   S706_TL_DC_3RD_CLAMP.Adv_End := TRUE;
   S706_TL_DC_3RD_CLAMP.Ret_End := FALSE;
   S706_TL_DC_U262_1_UP_DN.Enable_Aux := TRUE;
   S706_TL_DC_U262_1_UP_DN.Adv_Amount := 1;
   S706_TL_DC_U262_1_UP_DN.Ret_Amount := 1;
   S706_TL_DC_U262_1_UP_DN.LS_Adv1 := FALSE;
   S706_TL_DC_U262_1_UP_DN.LS_Ret1 := TRUE;
   S706_TL_DC_U262_1_UP_DN.LS_Adv2 := FALSE;
   S706_TL_DC_U262_1_UP_DN.LS_Ret2 := FALSE;
   S706_TL_DC_U262_1_UP_DN.LS_Adv3 := FALSE;
   S706_TL_DC_U262_1_UP_DN.LS_Ret3 := FALSE;
   S706_TL_DC_U262_1_UP_DN.LS_Adv4 := FALSE;
   S706_TL_DC_U262_1_UP_DN.LS_Ret4 := FALSE;
   S706_TL_DC_U262_1_UP_DN.LS_Adv5 := FALSE;
   S706_TL_DC_U262_1_UP_DN.LS_Ret5 := FALSE;
   S706_TL_DC_U262_1_UP_DN.LS_Adv6 := FALSE;
   S706_TL_DC_U262_1_UP_DN.LS_Ret6 := FALSE;
   S706_TL_DC_U262_1_UP_DN.LS_Adv7 := FALSE;
   S706_TL_DC_U262_1_UP_DN.LS_Ret7 := FALSE;
   S706_TL_DC_U262_1_UP_DN.LS_Adv8 := FALSE;
   S706_TL_DC_U262_1_UP_DN.LS_Ret8 := FALSE;
   S706_TL_DC_U262_1_UP_DN.SOL_Adv := FALSE;
   S706_TL_DC_U262_1_UP_DN.SOL_Ret := FALSE;
   S706_TL_DC_U262_1_UP_DN.M_Ready := TRUE;
   S706_TL_DC_U262_1_UP_DN.T_CHK1 := T#4S;
   S706_TL_DC_U262_1_UP_DN.T_CHK2 := T#4S;
   S706_TL_DC_U262_1_UP_DN.PB_Lamp_CHK := FALSE;
   S706_TL_DC_U262_1_UP_DN.PB_Error_Rst := FALSE;
   S706_TL_DC_U262_1_UP_DN.M_FLICK := FALSE;
   S706_TL_DC_U262_1_UP_DN.M_Adv_Err := FALSE;
   S706_TL_DC_U262_1_UP_DN.M_Ret_Err := FALSE;
   S706_TL_DC_U262_1_UP_DN.LP_Adv := FALSE;
   S706_TL_DC_U262_1_UP_DN.LP_Ret := TRUE;
   S706_TL_DC_U262_1_UP_DN.Visu_Adv := W#16#0;
   S706_TL_DC_U262_1_UP_DN.Visu_Ret := W#16#300;
   S706_TL_DC_U262_1_UP_DN.Error_T1.IN := FALSE;
   S706_TL_DC_U262_1_UP_DN.Error_T1.PT := T#4S;
   S706_TL_DC_U262_1_UP_DN.Error_T1.Q := FALSE;
   S706_TL_DC_U262_1_UP_DN.Error_T1.ET := T#0MS;
   S706_TL_DC_U262_1_UP_DN.Error_T1.STATE := B#16#0;
   S706_TL_DC_U262_1_UP_DN.Error_T1.STIME := T#23D5H8M21S546MS;
   S706_TL_DC_U262_1_UP_DN.Error_T1.ATIME := T#23D5H8M21S773MS;
   S706_TL_DC_U262_1_UP_DN.Error_T2.IN := FALSE;
   S706_TL_DC_U262_1_UP_DN.Error_T2.PT := T#4S;
   S706_TL_DC_U262_1_UP_DN.Error_T2.Q := FALSE;
   S706_TL_DC_U262_1_UP_DN.Error_T2.ET := T#0MS;
   S706_TL_DC_U262_1_UP_DN.Error_T2.STATE := B#16#0;
   S706_TL_DC_U262_1_UP_DN.Error_T2.STIME := T#0MS;
   S706_TL_DC_U262_1_UP_DN.Error_T2.ATIME := T#0MS;
   S706_TL_DC_U262_1_UP_DN.Adv_End_Aux := FALSE;
   S706_TL_DC_U262_1_UP_DN.Ret_End_Aux := TRUE;
   S706_TL_DC_U262_1_UP_DN.CHK_Aux1 := FALSE;
   S706_TL_DC_U262_1_UP_DN.CHK_Aux2 := FALSE;
   S706_TL_DC_U262_1_UP_DN.Error_T1_DN := FALSE;
   S706_TL_DC_U262_1_UP_DN.Error_T2_DN := FALSE;
   S706_TL_DC_U262_1_UP_DN.Adv_Memo := FALSE;
   S706_TL_DC_U262_1_UP_DN.Visu_Adv_Arr[0] := FALSE;
   S706_TL_DC_U262_1_UP_DN.Visu_Adv_Arr[1] := FALSE;
   S706_TL_DC_U262_1_UP_DN.Visu_Adv_Arr[2] := FALSE;
   S706_TL_DC_U262_1_UP_DN.Visu_Adv_Arr[3] := FALSE;
   S706_TL_DC_U262_1_UP_DN.Visu_Adv_Arr[4] := FALSE;
   S706_TL_DC_U262_1_UP_DN.Visu_Adv_Arr[5] := FALSE;
   S706_TL_DC_U262_1_UP_DN.Visu_Adv_Arr[6] := FALSE;
   S706_TL_DC_U262_1_UP_DN.Visu_Adv_Arr[7] := FALSE;
   S706_TL_DC_U262_1_UP_DN.Visu_Adv_Arr[8] := FALSE;
   S706_TL_DC_U262_1_UP_DN.Visu_Adv_Arr[9] := FALSE;
   S706_TL_DC_U262_1_UP_DN.Visu_Adv_Arr[10] := FALSE;
   S706_TL_DC_U262_1_UP_DN.Visu_Adv_Arr[11] := FALSE;
   S706_TL_DC_U262_1_UP_DN.Visu_Adv_Arr[12] := FALSE;
   S706_TL_DC_U262_1_UP_DN.Visu_Adv_Arr[13] := FALSE;
   S706_TL_DC_U262_1_UP_DN.Visu_Adv_Arr[14] := FALSE;
   S706_TL_DC_U262_1_UP_DN.Visu_Adv_Arr[15] := FALSE;
   S706_TL_DC_U262_1_UP_DN.Visu_Ret_Arr[0] := TRUE;
   S706_TL_DC_U262_1_UP_DN.Visu_Ret_Arr[1] := TRUE;
   S706_TL_DC_U262_1_UP_DN.Visu_Ret_Arr[2] := FALSE;
   S706_TL_DC_U262_1_UP_DN.Visu_Ret_Arr[3] := FALSE;
   S706_TL_DC_U262_1_UP_DN.Visu_Ret_Arr[4] := FALSE;
   S706_TL_DC_U262_1_UP_DN.Visu_Ret_Arr[5] := FALSE;
   S706_TL_DC_U262_1_UP_DN.Visu_Ret_Arr[6] := FALSE;
   S706_TL_DC_U262_1_UP_DN.Visu_Ret_Arr[7] := FALSE;
   S706_TL_DC_U262_1_UP_DN.Visu_Ret_Arr[8] := FALSE;
   S706_TL_DC_U262_1_UP_DN.Visu_Ret_Arr[9] := FALSE;
   S706_TL_DC_U262_1_UP_DN.Visu_Ret_Arr[10] := FALSE;
   S706_TL_DC_U262_1_UP_DN.Visu_Ret_Arr[11] := FALSE;
   S706_TL_DC_U262_1_UP_DN.Visu_Ret_Arr[12] := FALSE;
   S706_TL_DC_U262_1_UP_DN.Visu_Ret_Arr[13] := FALSE;
   S706_TL_DC_U262_1_UP_DN.Visu_Ret_Arr[14] := FALSE;
   S706_TL_DC_U262_1_UP_DN.Visu_Ret_Arr[15] := FALSE;
   S706_TL_DC_U262_1_UP_DN.BLK_Move_Ret := 0;
   S706_TL_DC_U262_1_UP_DN.Enable := TRUE;
   S706_TL_DC_U262_1_UP_DN.Adv_End := FALSE;
   S706_TL_DC_U262_1_UP_DN.Ret_End := TRUE;
   S706_TL_DC_U262_1.Enable_Aux := TRUE;
   S706_TL_DC_U262_1.Adv_Amount := 1;
   S706_TL_DC_U262_1.Ret_Amount := 1;
   S706_TL_DC_U262_1.LS_Adv1 := FALSE;
   S706_TL_DC_U262_1.LS_Ret1 := TRUE;
   S706_TL_DC_U262_1.LS_Adv2 := FALSE;
   S706_TL_DC_U262_1.LS_Ret2 := FALSE;
   S706_TL_DC_U262_1.LS_Adv3 := FALSE;
   S706_TL_DC_U262_1.LS_Ret3 := FALSE;
   S706_TL_DC_U262_1.LS_Adv4 := FALSE;
   S706_TL_DC_U262_1.LS_Ret4 := FALSE;
   S706_TL_DC_U262_1.LS_Adv5 := FALSE;
   S706_TL_DC_U262_1.LS_Ret5 := FALSE;
   S706_TL_DC_U262_1.LS_Adv6 := FALSE;
   S706_TL_DC_U262_1.LS_Ret6 := FALSE;
   S706_TL_DC_U262_1.LS_Adv7 := FALSE;
   S706_TL_DC_U262_1.LS_Ret7 := FALSE;
   S706_TL_DC_U262_1.LS_Adv8 := FALSE;
   S706_TL_DC_U262_1.LS_Ret8 := FALSE;
   S706_TL_DC_U262_1.SOL_Adv := FALSE;
   S706_TL_DC_U262_1.SOL_Ret := FALSE;
   S706_TL_DC_U262_1.M_Ready := TRUE;
   S706_TL_DC_U262_1.T_CHK1 := T#4S;
   S706_TL_DC_U262_1.T_CHK2 := T#4S;
   S706_TL_DC_U262_1.PB_Lamp_CHK := FALSE;
   S706_TL_DC_U262_1.PB_Error_Rst := FALSE;
   S706_TL_DC_U262_1.M_FLICK := FALSE;
   S706_TL_DC_U262_1.M_Adv_Err := FALSE;
   S706_TL_DC_U262_1.M_Ret_Err := FALSE;
   S706_TL_DC_U262_1.LP_Adv := FALSE;
   S706_TL_DC_U262_1.LP_Ret := TRUE;
   S706_TL_DC_U262_1.Visu_Adv := W#16#0;
   S706_TL_DC_U262_1.Visu_Ret := W#16#300;
   S706_TL_DC_U262_1.Error_T1.IN := FALSE;
   S706_TL_DC_U262_1.Error_T1.PT := T#4S;
   S706_TL_DC_U262_1.Error_T1.Q := FALSE;
   S706_TL_DC_U262_1.Error_T1.ET := T#0MS;
   S706_TL_DC_U262_1.Error_T1.STATE := B#16#0;
   S706_TL_DC_U262_1.Error_T1.STIME := T#23D2H56M52S237MS;
   S706_TL_DC_U262_1.Error_T1.ATIME := T#23D2H56M52S283MS;
   S706_TL_DC_U262_1.Error_T2.IN := FALSE;
   S706_TL_DC_U262_1.Error_T2.PT := T#4S;
   S706_TL_DC_U262_1.Error_T2.Q := FALSE;
   S706_TL_DC_U262_1.Error_T2.ET := T#0MS;
   S706_TL_DC_U262_1.Error_T2.STATE := B#16#0;
   S706_TL_DC_U262_1.Error_T2.STIME := T#0MS;
   S706_TL_DC_U262_1.Error_T2.ATIME := T#0MS;
   S706_TL_DC_U262_1.Adv_End_Aux := FALSE;
   S706_TL_DC_U262_1.Ret_End_Aux := TRUE;
   S706_TL_DC_U262_1.CHK_Aux1 := FALSE;
   S706_TL_DC_U262_1.CHK_Aux2 := FALSE;
   S706_TL_DC_U262_1.Error_T1_DN := FALSE;
   S706_TL_DC_U262_1.Error_T2_DN := FALSE;
   S706_TL_DC_U262_1.Adv_Memo := FALSE;
   S706_TL_DC_U262_1.Visu_Adv_Arr[0] := FALSE;
   S706_TL_DC_U262_1.Visu_Adv_Arr[1] := FALSE;
   S706_TL_DC_U262_1.Visu_Adv_Arr[2] := FALSE;
   S706_TL_DC_U262_1.Visu_Adv_Arr[3] := FALSE;
   S706_TL_DC_U262_1.Visu_Adv_Arr[4] := FALSE;
   S706_TL_DC_U262_1.Visu_Adv_Arr[5] := FALSE;
   S706_TL_DC_U262_1.Visu_Adv_Arr[6] := FALSE;
   S706_TL_DC_U262_1.Visu_Adv_Arr[7] := FALSE;
   S706_TL_DC_U262_1.Visu_Adv_Arr[8] := FALSE;
   S706_TL_DC_U262_1.Visu_Adv_Arr[9] := FALSE;
   S706_TL_DC_U262_1.Visu_Adv_Arr[10] := FALSE;
   S706_TL_DC_U262_1.Visu_Adv_Arr[11] := FALSE;
   S706_TL_DC_U262_1.Visu_Adv_Arr[12] := FALSE;
   S706_TL_DC_U262_1.Visu_Adv_Arr[13] := FALSE;
   S706_TL_DC_U262_1.Visu_Adv_Arr[14] := FALSE;
   S706_TL_DC_U262_1.Visu_Adv_Arr[15] := FALSE;
   S706_TL_DC_U262_1.Visu_Ret_Arr[0] := TRUE;
   S706_TL_DC_U262_1.Visu_Ret_Arr[1] := TRUE;
   S706_TL_DC_U262_1.Visu_Ret_Arr[2] := FALSE;
   S706_TL_DC_U262_1.Visu_Ret_Arr[3] := FALSE;
   S706_TL_DC_U262_1.Visu_Ret_Arr[4] := FALSE;
   S706_TL_DC_U262_1.Visu_Ret_Arr[5] := FALSE;
   S706_TL_DC_U262_1.Visu_Ret_Arr[6] := FALSE;
   S706_TL_DC_U262_1.Visu_Ret_Arr[7] := FALSE;
   S706_TL_DC_U262_1.Visu_Ret_Arr[8] := FALSE;
   S706_TL_DC_U262_1.Visu_Ret_Arr[9] := FALSE;
   S706_TL_DC_U262_1.Visu_Ret_Arr[10] := FALSE;
   S706_TL_DC_U262_1.Visu_Ret_Arr[11] := FALSE;
   S706_TL_DC_U262_1.Visu_Ret_Arr[12] := FALSE;
   S706_TL_DC_U262_1.Visu_Ret_Arr[13] := FALSE;
   S706_TL_DC_U262_1.Visu_Ret_Arr[14] := FALSE;
   S706_TL_DC_U262_1.Visu_Ret_Arr[15] := FALSE;
   S706_TL_DC_U262_1.BLK_Move_Ret := 0;
   S706_TL_DC_U262_1.Enable := TRUE;
   S706_TL_DC_U262_1.Adv_End := FALSE;
   S706_TL_DC_U262_1.Ret_End := TRUE;
   S706_TL_DC_U262_1_CLAMP.Enable_Aux := TRUE;
   S706_TL_DC_U262_1_CLAMP.Adv_Amount := 1;
   S706_TL_DC_U262_1_CLAMP.Ret_Amount := 1;
   S706_TL_DC_U262_1_CLAMP.LS_Adv1 := FALSE;
   S706_TL_DC_U262_1_CLAMP.LS_Ret1 := TRUE;
   S706_TL_DC_U262_1_CLAMP.LS_Adv2 := FALSE;
   S706_TL_DC_U262_1_CLAMP.LS_Ret2 := FALSE;
   S706_TL_DC_U262_1_CLAMP.LS_Adv3 := FALSE;
   S706_TL_DC_U262_1_CLAMP.LS_Ret3 := FALSE;
   S706_TL_DC_U262_1_CLAMP.LS_Adv4 := FALSE;
   S706_TL_DC_U262_1_CLAMP.LS_Ret4 := FALSE;
   S706_TL_DC_U262_1_CLAMP.LS_Adv5 := FALSE;
   S706_TL_DC_U262_1_CLAMP.LS_Ret5 := FALSE;
   S706_TL_DC_U262_1_CLAMP.LS_Adv6 := FALSE;
   S706_TL_DC_U262_1_CLAMP.LS_Ret6 := FALSE;
   S706_TL_DC_U262_1_CLAMP.LS_Adv7 := FALSE;
   S706_TL_DC_U262_1_CLAMP.LS_Ret7 := FALSE;
   S706_TL_DC_U262_1_CLAMP.LS_Adv8 := FALSE;
   S706_TL_DC_U262_1_CLAMP.LS_Ret8 := FALSE;
   S706_TL_DC_U262_1_CLAMP.SOL_Adv := FALSE;
   S706_TL_DC_U262_1_CLAMP.SOL_Ret := FALSE;
   S706_TL_DC_U262_1_CLAMP.M_Ready := TRUE;
   S706_TL_DC_U262_1_CLAMP.T_CHK1 := T#4S;
   S706_TL_DC_U262_1_CLAMP.T_CHK2 := T#4S;
   S706_TL_DC_U262_1_CLAMP.PB_Lamp_CHK := FALSE;
   S706_TL_DC_U262_1_CLAMP.PB_Error_Rst := FALSE;
   S706_TL_DC_U262_1_CLAMP.M_FLICK := FALSE;
   S706_TL_DC_U262_1_CLAMP.M_Adv_Err := FALSE;
   S706_TL_DC_U262_1_CLAMP.M_Ret_Err := FALSE;
   S706_TL_DC_U262_1_CLAMP.LP_Adv := FALSE;
   S706_TL_DC_U262_1_CLAMP.LP_Ret := TRUE;
   S706_TL_DC_U262_1_CLAMP.Visu_Adv := W#16#0;
   S706_TL_DC_U262_1_CLAMP.Visu_Ret := W#16#300;
   S706_TL_DC_U262_1_CLAMP.Error_T1.IN := FALSE;
   S706_TL_DC_U262_1_CLAMP.Error_T1.PT := T#4S;
   S706_TL_DC_U262_1_CLAMP.Error_T1.Q := FALSE;
   S706_TL_DC_U262_1_CLAMP.Error_T1.ET := T#0MS;
   S706_TL_DC_U262_1_CLAMP.Error_T1.STATE := B#16#0;
   S706_TL_DC_U262_1_CLAMP.Error_T1.STIME := T#23D2H56M52S237MS;
   S706_TL_DC_U262_1_CLAMP.Error_T1.ATIME := T#23D2H56M52S283MS;
   S706_TL_DC_U262_1_CLAMP.Error_T2.IN := FALSE;
   S706_TL_DC_U262_1_CLAMP.Error_T2.PT := T#4S;
   S706_TL_DC_U262_1_CLAMP.Error_T2.Q := FALSE;
   S706_TL_DC_U262_1_CLAMP.Error_T2.ET := T#0MS;
   S706_TL_DC_U262_1_CLAMP.Error_T2.STATE := B#16#0;
   S706_TL_DC_U262_1_CLAMP.Error_T2.STIME := T#0MS;
   S706_TL_DC_U262_1_CLAMP.Error_T2.ATIME := T#0MS;
   S706_TL_DC_U262_1_CLAMP.Adv_End_Aux := FALSE;
   S706_TL_DC_U262_1_CLAMP.Ret_End_Aux := TRUE;
   S706_TL_DC_U262_1_CLAMP.CHK_Aux1 := FALSE;
   S706_TL_DC_U262_1_CLAMP.CHK_Aux2 := FALSE;
   S706_TL_DC_U262_1_CLAMP.Error_T1_DN := FALSE;
   S706_TL_DC_U262_1_CLAMP.Error_T2_DN := FALSE;
   S706_TL_DC_U262_1_CLAMP.Adv_Memo := FALSE;
   S706_TL_DC_U262_1_CLAMP.Visu_Adv_Arr[0] := FALSE;
   S706_TL_DC_U262_1_CLAMP.Visu_Adv_Arr[1] := FALSE;
   S706_TL_DC_U262_1_CLAMP.Visu_Adv_Arr[2] := FALSE;
   S706_TL_DC_U262_1_CLAMP.Visu_Adv_Arr[3] := FALSE;
   S706_TL_DC_U262_1_CLAMP.Visu_Adv_Arr[4] := FALSE;
   S706_TL_DC_U262_1_CLAMP.Visu_Adv_Arr[5] := FALSE;
   S706_TL_DC_U262_1_CLAMP.Visu_Adv_Arr[6] := FALSE;
   S706_TL_DC_U262_1_CLAMP.Visu_Adv_Arr[7] := FALSE;
   S706_TL_DC_U262_1_CLAMP.Visu_Adv_Arr[8] := FALSE;
   S706_TL_DC_U262_1_CLAMP.Visu_Adv_Arr[9] := FALSE;
   S706_TL_DC_U262_1_CLAMP.Visu_Adv_Arr[10] := FALSE;
   S706_TL_DC_U262_1_CLAMP.Visu_Adv_Arr[11] := FALSE;
   S706_TL_DC_U262_1_CLAMP.Visu_Adv_Arr[12] := FALSE;
   S706_TL_DC_U262_1_CLAMP.Visu_Adv_Arr[13] := FALSE;
   S706_TL_DC_U262_1_CLAMP.Visu_Adv_Arr[14] := FALSE;
   S706_TL_DC_U262_1_CLAMP.Visu_Adv_Arr[15] := FALSE;
   S706_TL_DC_U262_1_CLAMP.Visu_Ret_Arr[0] := TRUE;
   S706_TL_DC_U262_1_CLAMP.Visu_Ret_Arr[1] := TRUE;
   S706_TL_DC_U262_1_CLAMP.Visu_Ret_Arr[2] := FALSE;
   S706_TL_DC_U262_1_CLAMP.Visu_Ret_Arr[3] := FALSE;
   S706_TL_DC_U262_1_CLAMP.Visu_Ret_Arr[4] := FALSE;
   S706_TL_DC_U262_1_CLAMP.Visu_Ret_Arr[5] := FALSE;
   S706_TL_DC_U262_1_CLAMP.Visu_Ret_Arr[6] := FALSE;
   S706_TL_DC_U262_1_CLAMP.Visu_Ret_Arr[7] := FALSE;
   S706_TL_DC_U262_1_CLAMP.Visu_Ret_Arr[8] := FALSE;
   S706_TL_DC_U262_1_CLAMP.Visu_Ret_Arr[9] := FALSE;
   S706_TL_DC_U262_1_CLAMP.Visu_Ret_Arr[10] := FALSE;
   S706_TL_DC_U262_1_CLAMP.Visu_Ret_Arr[11] := FALSE;
   S706_TL_DC_U262_1_CLAMP.Visu_Ret_Arr[12] := FALSE;
   S706_TL_DC_U262_1_CLAMP.Visu_Ret_Arr[13] := FALSE;
   S706_TL_DC_U262_1_CLAMP.Visu_Ret_Arr[14] := FALSE;
   S706_TL_DC_U262_1_CLAMP.Visu_Ret_Arr[15] := FALSE;
   S706_TL_DC_U262_1_CLAMP.BLK_Move_Ret := 0;
   S706_TL_DC_U262_1_CLAMP.Enable := TRUE;
   S706_TL_DC_U262_1_CLAMP.Adv_End := FALSE;
   S706_TL_DC_U262_1_CLAMP.Ret_End := TRUE;
   S706_TL_DC_U261_2_CLAMP.Enable_Aux := TRUE;
   S706_TL_DC_U261_2_CLAMP.Adv_Amount := 1;
   S706_TL_DC_U261_2_CLAMP.Ret_Amount := 1;
   S706_TL_DC_U261_2_CLAMP.LS_Adv1 := FALSE;
   S706_TL_DC_U261_2_CLAMP.LS_Ret1 := TRUE;
   S706_TL_DC_U261_2_CLAMP.LS_Adv2 := FALSE;
   S706_TL_DC_U261_2_CLAMP.LS_Ret2 := FALSE;
   S706_TL_DC_U261_2_CLAMP.LS_Adv3 := FALSE;
   S706_TL_DC_U261_2_CLAMP.LS_Ret3 := FALSE;
   S706_TL_DC_U261_2_CLAMP.LS_Adv4 := FALSE;
   S706_TL_DC_U261_2_CLAMP.LS_Ret4 := FALSE;
   S706_TL_DC_U261_2_CLAMP.LS_Adv5 := FALSE;
   S706_TL_DC_U261_2_CLAMP.LS_Ret5 := FALSE;
   S706_TL_DC_U261_2_CLAMP.LS_Adv6 := FALSE;
   S706_TL_DC_U261_2_CLAMP.LS_Ret6 := FALSE;
   S706_TL_DC_U261_2_CLAMP.LS_Adv7 := FALSE;
   S706_TL_DC_U261_2_CLAMP.LS_Ret7 := FALSE;
   S706_TL_DC_U261_2_CLAMP.LS_Adv8 := FALSE;
   S706_TL_DC_U261_2_CLAMP.LS_Ret8 := FALSE;
   S706_TL_DC_U261_2_CLAMP.SOL_Adv := FALSE;
   S706_TL_DC_U261_2_CLAMP.SOL_Ret := FALSE;
   S706_TL_DC_U261_2_CLAMP.M_Ready := TRUE;
   S706_TL_DC_U261_2_CLAMP.T_CHK1 := T#4S;
   S706_TL_DC_U261_2_CLAMP.T_CHK2 := T#4S;
   S706_TL_DC_U261_2_CLAMP.PB_Lamp_CHK := FALSE;
   S706_TL_DC_U261_2_CLAMP.PB_Error_Rst := FALSE;
   S706_TL_DC_U261_2_CLAMP.M_FLICK := FALSE;
   S706_TL_DC_U261_2_CLAMP.M_Adv_Err := FALSE;
   S706_TL_DC_U261_2_CLAMP.M_Ret_Err := FALSE;
   S706_TL_DC_U261_2_CLAMP.LP_Adv := FALSE;
   S706_TL_DC_U261_2_CLAMP.LP_Ret := TRUE;
   S706_TL_DC_U261_2_CLAMP.Visu_Adv := W#16#0;
   S706_TL_DC_U261_2_CLAMP.Visu_Ret := W#16#300;
   S706_TL_DC_U261_2_CLAMP.Error_T1.IN := FALSE;
   S706_TL_DC_U261_2_CLAMP.Error_T1.PT := T#4S;
   S706_TL_DC_U261_2_CLAMP.Error_T1.Q := FALSE;
   S706_TL_DC_U261_2_CLAMP.Error_T1.ET := T#0MS;
   S706_TL_DC_U261_2_CLAMP.Error_T1.STATE := B#16#0;
   S706_TL_DC_U261_2_CLAMP.Error_T1.STIME := T#23D5H7M6S627MS;
   S706_TL_DC_U261_2_CLAMP.Error_T1.ATIME := T#23D5H7M6S855MS;
   S706_TL_DC_U261_2_CLAMP.Error_T2.IN := FALSE;
   S706_TL_DC_U261_2_CLAMP.Error_T2.PT := T#4S;
   S706_TL_DC_U261_2_CLAMP.Error_T2.Q := FALSE;
   S706_TL_DC_U261_2_CLAMP.Error_T2.ET := T#0MS;
   S706_TL_DC_U261_2_CLAMP.Error_T2.STATE := B#16#0;
   S706_TL_DC_U261_2_CLAMP.Error_T2.STIME := T#23D5H7M45S906MS;
   S706_TL_DC_U261_2_CLAMP.Error_T2.ATIME := T#23D5H7M45S953MS;
   S706_TL_DC_U261_2_CLAMP.Adv_End_Aux := FALSE;
   S706_TL_DC_U261_2_CLAMP.Ret_End_Aux := TRUE;
   S706_TL_DC_U261_2_CLAMP.CHK_Aux1 := FALSE;
   S706_TL_DC_U261_2_CLAMP.CHK_Aux2 := FALSE;
   S706_TL_DC_U261_2_CLAMP.Error_T1_DN := FALSE;
   S706_TL_DC_U261_2_CLAMP.Error_T2_DN := FALSE;
   S706_TL_DC_U261_2_CLAMP.Adv_Memo := FALSE;
   S706_TL_DC_U261_2_CLAMP.Visu_Adv_Arr[0] := FALSE;
   S706_TL_DC_U261_2_CLAMP.Visu_Adv_Arr[1] := FALSE;
   S706_TL_DC_U261_2_CLAMP.Visu_Adv_Arr[2] := FALSE;
   S706_TL_DC_U261_2_CLAMP.Visu_Adv_Arr[3] := FALSE;
   S706_TL_DC_U261_2_CLAMP.Visu_Adv_Arr[4] := FALSE;
   S706_TL_DC_U261_2_CLAMP.Visu_Adv_Arr[5] := FALSE;
   S706_TL_DC_U261_2_CLAMP.Visu_Adv_Arr[6] := FALSE;
   S706_TL_DC_U261_2_CLAMP.Visu_Adv_Arr[7] := FALSE;
   S706_TL_DC_U261_2_CLAMP.Visu_Adv_Arr[8] := FALSE;
   S706_TL_DC_U261_2_CLAMP.Visu_Adv_Arr[9] := FALSE;
   S706_TL_DC_U261_2_CLAMP.Visu_Adv_Arr[10] := FALSE;
   S706_TL_DC_U261_2_CLAMP.Visu_Adv_Arr[11] := FALSE;
   S706_TL_DC_U261_2_CLAMP.Visu_Adv_Arr[12] := FALSE;
   S706_TL_DC_U261_2_CLAMP.Visu_Adv_Arr[13] := FALSE;
   S706_TL_DC_U261_2_CLAMP.Visu_Adv_Arr[14] := FALSE;
   S706_TL_DC_U261_2_CLAMP.Visu_Adv_Arr[15] := FALSE;
   S706_TL_DC_U261_2_CLAMP.Visu_Ret_Arr[0] := TRUE;
   S706_TL_DC_U261_2_CLAMP.Visu_Ret_Arr[1] := TRUE;
   S706_TL_DC_U261_2_CLAMP.Visu_Ret_Arr[2] := FALSE;
   S706_TL_DC_U261_2_CLAMP.Visu_Ret_Arr[3] := FALSE;
   S706_TL_DC_U261_2_CLAMP.Visu_Ret_Arr[4] := FALSE;
   S706_TL_DC_U261_2_CLAMP.Visu_Ret_Arr[5] := FALSE;
   S706_TL_DC_U261_2_CLAMP.Visu_Ret_Arr[6] := FALSE;
   S706_TL_DC_U261_2_CLAMP.Visu_Ret_Arr[7] := FALSE;
   S706_TL_DC_U261_2_CLAMP.Visu_Ret_Arr[8] := FALSE;
   S706_TL_DC_U261_2_CLAMP.Visu_Ret_Arr[9] := FALSE;
   S706_TL_DC_U261_2_CLAMP.Visu_Ret_Arr[10] := FALSE;
   S706_TL_DC_U261_2_CLAMP.Visu_Ret_Arr[11] := FALSE;
   S706_TL_DC_U261_2_CLAMP.Visu_Ret_Arr[12] := FALSE;
   S706_TL_DC_U261_2_CLAMP.Visu_Ret_Arr[13] := FALSE;
   S706_TL_DC_U261_2_CLAMP.Visu_Ret_Arr[14] := FALSE;
   S706_TL_DC_U261_2_CLAMP.Visu_Ret_Arr[15] := FALSE;
   S706_TL_DC_U261_2_CLAMP.BLK_Move_Ret := 0;
   S706_TL_DC_U261_2_CLAMP.Enable := TRUE;
   S706_TL_DC_U261_2_CLAMP.Adv_End := FALSE;
   S706_TL_DC_U261_2_CLAMP.Ret_End := TRUE;
END_DATA_BLOCK

FUNCTION FC 124 : VOID
TITLE =
VERSION : 0.1

BEGIN
NETWORK
TITLE =
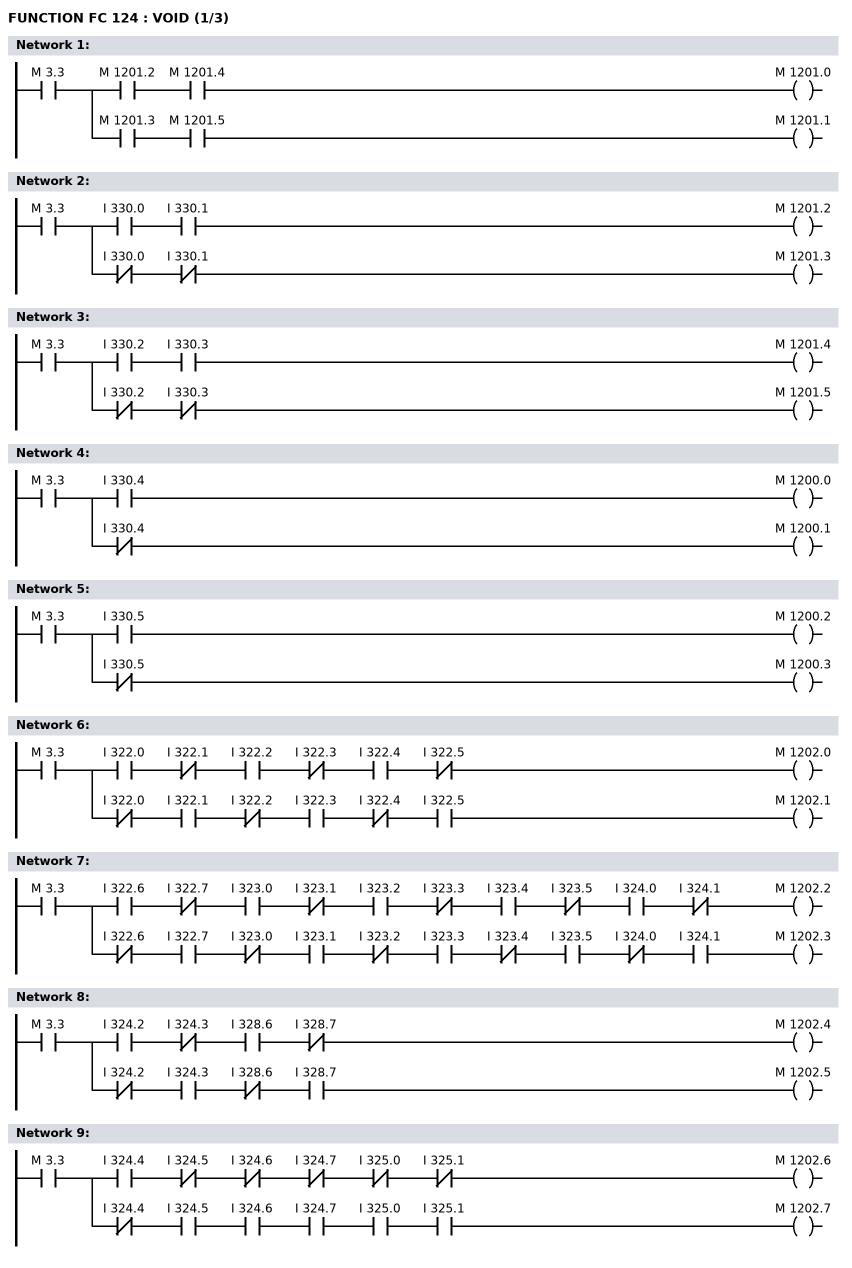

      A     M      3.3;
      =     L      0.0;
      A     L      0.0;
      A     M   1201.2;
      A     M   1201.4;
      =     M   1201.0;
      A     L      0.0;
      A     M   1201.3;
      A     M   1201.5;
      =     M   1201.1;
NETWORK
TITLE =

      A     M      3.3;
      =     L      0.0;
      A     L      0.0;
      A     I    330.0;
      A     I    330.1;
      =     M   1201.2;
      A     L      0.0;
      AN    I    330.0;
      AN    I    330.1;
      =     M   1201.3;
NETWORK
TITLE =

      A     M      3.3;
      =     L      0.0;
      A     L      0.0;
      A     I    330.2;
      A     I    330.3;
      =     M   1201.4;
      A     L      0.0;
      AN    I    330.2;
      AN    I    330.3;
      =     M   1201.5;
NETWORK
TITLE =

      A     M      3.3;
      =     L      0.0;
      A     L      0.0;
      A     I    330.4;
      =     M   1200.0;
      A     L      0.0;
      AN    I    330.4;
      =     M   1200.1;
NETWORK
TITLE =

      A     M      3.3;
      =     L      0.0;
      A     L      0.0;
      A     I    330.5;
      =     M   1200.2;
      A     L      0.0;
      AN    I    330.5;
      =     M   1200.3;
NETWORK
TITLE =

      A     M      3.3;
      =     L      0.0;
      A     L      0.0;
      A     I    322.0;
      AN    I    322.1;
      A     I    322.2;
      AN    I    322.3;
      A     I    322.4;
      AN    I    322.5;
      =     M   1202.0;
      A     L      0.0;
      AN    I    322.0;
      A     I    322.1;
      AN    I    322.2;
      A     I    322.3;
      AN    I    322.4;
      A     I    322.5;
      =     M   1202.1;
NETWORK
TITLE =

      A     M      3.3;
      =     L      0.0;
      A     L      0.0;
      A     I    322.6;
      AN    I    322.7;
      A     I    323.0;
      AN    I    323.1;
      A     I    323.2;
      AN    I    323.3;
      A     I    323.4;
      AN    I    323.5;
      A     I    324.0;
      AN    I    324.1;
      =     M   1202.2;
      A     L      0.0;
      AN    I    322.6;
      A     I    322.7;
      AN    I    323.0;
      A     I    323.1;
      AN    I    323.2;
      A     I    323.3;
      AN    I    323.4;
      A     I    323.5;
      AN    I    324.0;
      A     I    324.1;
      =     M   1202.3;
NETWORK
TITLE =

      A     M      3.3;
      =     L      0.0;
      A     L      0.0;
      A     I    324.2;
      AN    I    324.3;
      A     I    328.6;
      AN    I    328.7;
      =     M   1202.4;
      A     L      0.0;
      AN    I    324.2;
      A     I    324.3;
      AN    I    328.6;
      A     I    328.7;
      =     M   1202.5;
NETWORK
TITLE =

      A     M      3.3;
      =     L      0.0;
      A     L      0.0;
      A     I    324.4;
      AN    I    324.5;
      AN    I    324.6;
      AN    I    324.7;
      AN    I    325.0;
      AN    I    325.1;
      =     M   1202.6;
      A     L      0.0;
      AN    I    324.4;
      A     I    324.5;
      A     I    324.6;
      A     I    324.7;
      A     I    325.0;
      A     I    325.1;
      =     M   1202.7;
NETWORK
TITLE =
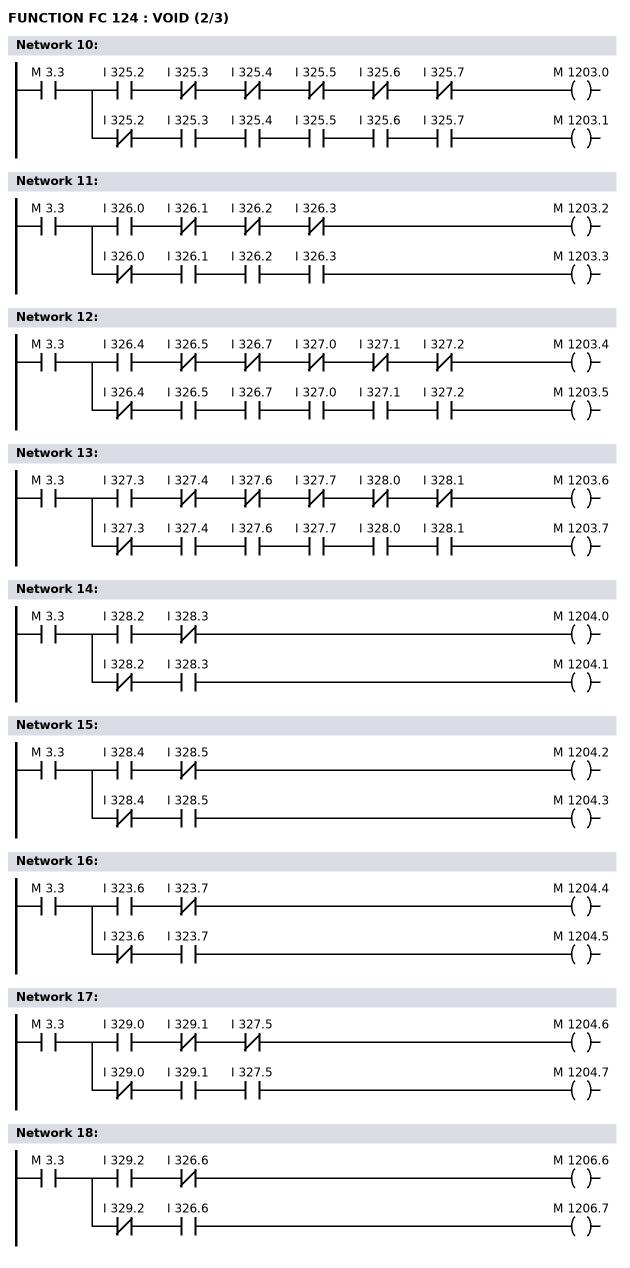

      A     M      3.3;
      =     L      0.0;
      A     L      0.0;
      A     I    325.2;
      AN    I    325.3;
      AN    I    325.4;
      AN    I    325.5;
      AN    I    325.6;
      AN    I    325.7;
      =     M   1203.0;
      A     L      0.0;
      AN    I    325.2;
      A     I    325.3;
      A     I    325.4;
      A     I    325.5;
      A     I    325.6;
      A     I    325.7;
      =     M   1203.1;
NETWORK
TITLE =

      A     M      3.3;
      =     L      0.0;
      A     L      0.0;
      A     I    326.0;
      AN    I    326.1;
      AN    I    326.2;
      AN    I    326.3;
      =     M   1203.2;
      A     L      0.0;
      AN    I    326.0;
      A     I    326.1;
      A     I    326.2;
      A     I    326.3;
      =     M   1203.3;
NETWORK
TITLE =

      A     M      3.3;
      =     L      0.0;
      A     L      0.0;
      A     I    326.4;
      AN    I    326.5;
      AN    I    326.7;
      AN    I    327.0;
      AN    I    327.1;
      AN    I    327.2;
      =     M   1203.4;
      A     L      0.0;
      AN    I    326.4;
      A     I    326.5;
      A     I    326.7;
      A     I    327.0;
      A     I    327.1;
      A     I    327.2;
      =     M   1203.5;
NETWORK
TITLE =

      A     M      3.3;
      =     L      0.0;
      A     L      0.0;
      A     I    327.3;
      AN    I    327.4;
      AN    I    327.6;
      AN    I    327.7;
      AN    I    328.0;
      AN    I    328.1;
      =     M   1203.6;
      A     L      0.0;
      AN    I    327.3;
      A     I    327.4;
      A     I    327.6;
      A     I    327.7;
      A     I    328.0;
      A     I    328.1;
      =     M   1203.7;
NETWORK
TITLE =

      A     M      3.3;
      =     L      0.0;
      A     L      0.0;
      A     I    328.2;
      AN    I    328.3;
      =     M   1204.0;
      A     L      0.0;
      AN    I    328.2;
      A     I    328.3;
      =     M   1204.1;
NETWORK
TITLE =

      A     M      3.3;
      =     L      0.0;
      A     L      0.0;
      A     I    328.4;
      AN    I    328.5;
      =     M   1204.2;
      A     L      0.0;
      AN    I    328.4;
      A     I    328.5;
      =     M   1204.3;
NETWORK
TITLE =

      A     M      3.3;
      =     L      0.0;
      A     L      0.0;
      A     I    323.6;
      AN    I    323.7;
      =     M   1204.4;
      A     L      0.0;
      AN    I    323.6;
      A     I    323.7;
      =     M   1204.5;
NETWORK
TITLE =

      A     M      3.3;
      =     L      0.0;
      A     L      0.0;
      A     I    329.0;
      AN    I    329.1;
      AN    I    327.5;
      =     M   1204.6;
      A     L      0.0;
      AN    I    329.0;
      A     I    329.1;
      A     I    327.5;
      =     M   1204.7;
NETWORK
TITLE =

      A     M      3.3;
      =     L      0.0;
      A     L      0.0;
      A     I    329.2;
      AN    I    326.6;
      =     M   1206.6;
      A     L      0.0;
      AN    I    329.2;
      A     I    326.6;
      =     M   1206.7;
NETWORK
TITLE =
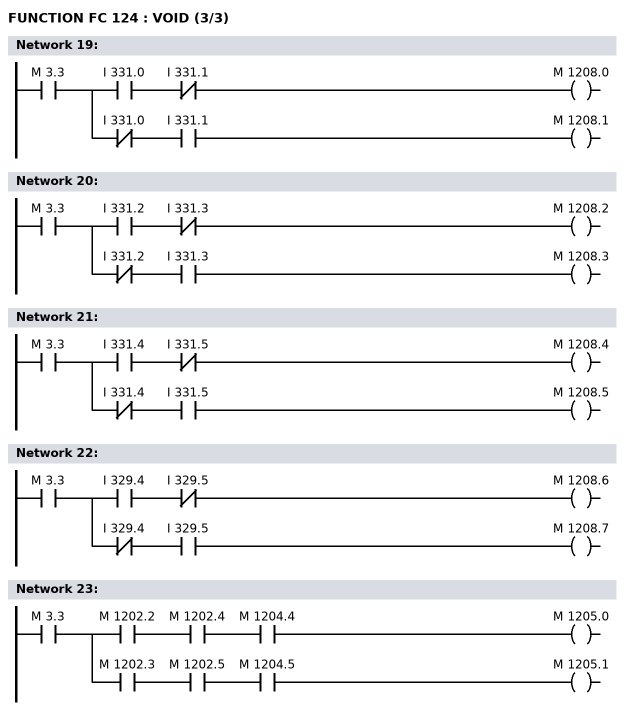

      A     M      3.3;
      =     L      0.0;
      A     L      0.0;
      A     I    331.0;
      AN    I    331.1;
      =     M   1208.0;
      A     L      0.0;
      AN    I    331.0;
      A     I    331.1;
      =     M   1208.1;
NETWORK
TITLE =

      A     M      3.3;
      =     L      0.0;
      A     L      0.0;
      A     I    331.2;
      AN    I    331.3;
      =     M   1208.2;
      A     L      0.0;
      AN    I    331.2;
      A     I    331.3;
      =     M   1208.3;
NETWORK
TITLE =

      A     M      3.3;
      =     L      0.0;
      A     L      0.0;
      A     I    331.4;
      AN    I    331.5;
      =     M   1208.4;
      A     L      0.0;
      AN    I    331.4;
      A     I    331.5;
      =     M   1208.5;
NETWORK
TITLE =

      A     M      3.3;
      =     L      0.0;
      A     L      0.0;
      A     I    329.4;
      AN    I    329.5;
      =     M   1208.6;
      A     L      0.0;
      AN    I    329.4;
      A     I    329.5;
      =     M   1208.7;
NETWORK
TITLE =

      A     M      3.3;
      =     L      0.0;
      A     L      0.0;
      A     M   1202.2;
      A     M   1202.4;
      A     M   1204.4;
      =     M   1205.0;
      A     L      0.0;
      A     M   1202.3;
      A     M   1202.5;
      A     M   1204.5;
      =     M   1205.1;
NETWORK
TITLE =

      A     M      3.3;
      =     L      0.0;
      A     L      0.0;
      A     M   1202.6;
      A     M   1203.0;
      A     M   1203.2;
      A     M   1203.4;
      A     M   1203.6;
      A     M   1206.6;
      =     L      0.1;
      A     L      0.1;
      BLD   102;
      =     M   1205.2;
      A     L      0.1;
      A     M   1204.2;
      A     M   1204.6;
      =     M   1205.4;
      A     L      0.0;
      A     M   1202.7;
      A     M   1203.1;
      A     M   1203.3;
      A     M   1203.5;
      A     M   1203.7;
      A     M   1206.7;
      =     L      0.1;
      A     L      0.1;
      BLD   102;
      =     M   1205.3;
      A     L      0.1;
      A     M   1204.3;
      A     M   1204.7;
      =     M   1205.5;
NETWORK
TITLE =
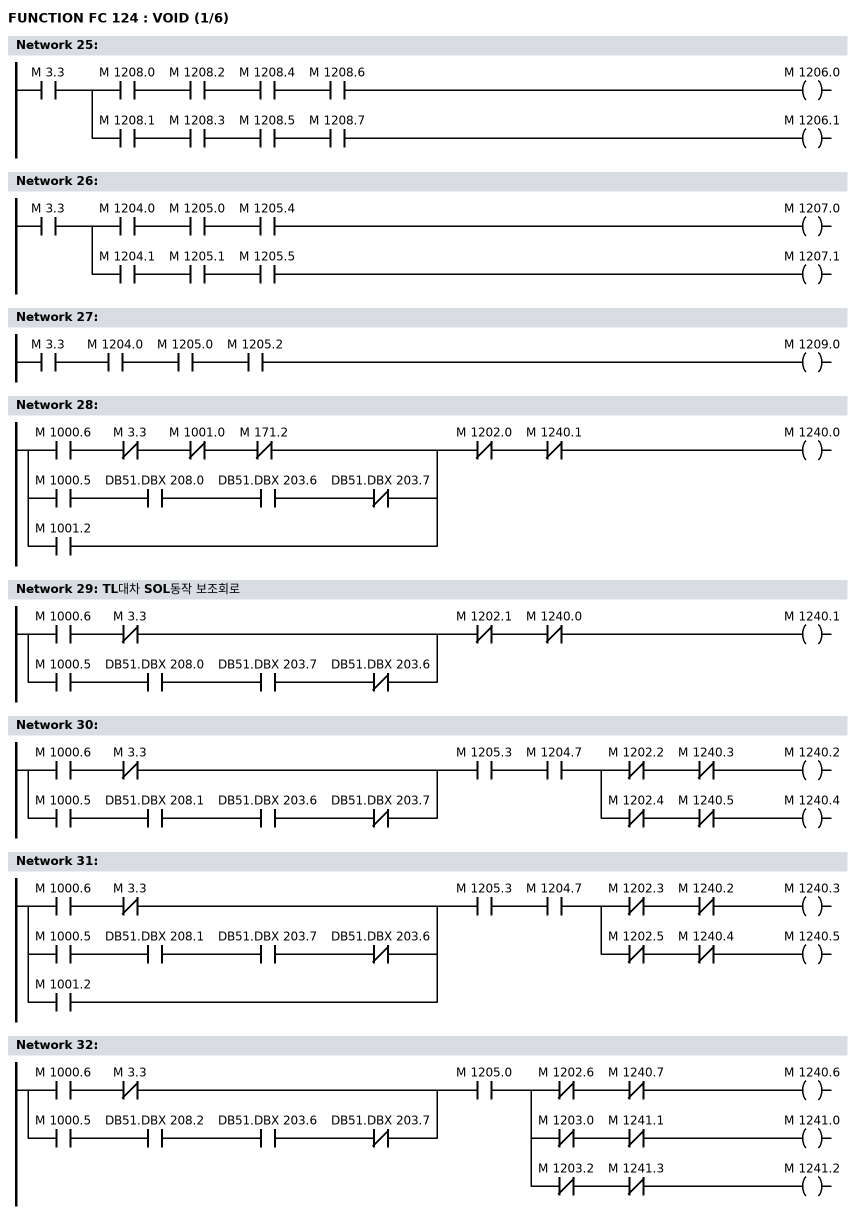

      A     M      3.3;
      =     L      0.0;
      A     L      0.0;
      A     M   1208.0;
      A     M   1208.2;
      A     M   1208.4;
      A     M   1208.6;
      =     M   1206.0;
      A     L      0.0;
      A     M   1208.1;
      A     M   1208.3;
      A     M   1208.5;
      A     M   1208.7;
      =     M   1206.1;
NETWORK
TITLE =

      A     M      3.3;
      =     L      0.0;
      A     L      0.0;
      A     M   1204.0;
      A     M   1205.0;
      A     M   1205.4;
      =     M   1207.0;
      A     L      0.0;
      A     M   1204.1;
      A     M   1205.1;
      A     M   1205.5;
      =     M   1207.1;
NETWORK
TITLE =

      A     M      3.3;
      A     M   1204.0;
      A     M   1205.0;
      A     M   1205.2;
      =     M   1209.0;
NETWORK
TITLE =

      A(    ;
      A     M   1000.6;
      AN    M      3.3;
      AN    M   1001.0;
      AN    M    171.2;
      O     ;
      A     M   1000.5;
      A     DB51.DBX  208.0;
      A     DB51.DBX  203.6;
      AN    DB51.DBX  203.7;
      O     M   1001.2;
      )     ;
      AN    M   1202.0;
      AN    M   1240.1;
      =     M   1240.0;
NETWORK
TITLE =TL대차 SOL동작 보조회로

      A(    ;
      A     M   1000.6;
      AN    M      3.3;
      O     ;
      A     M   1000.5;
      A     DB51.DBX  208.0;
      A     DB51.DBX  203.7;
      AN    DB51.DBX  203.6;
      )     ;
      AN    M   1202.1;
      AN    M   1240.0;
      =     M   1240.1;
NETWORK
TITLE =

      A(    ;
      A     M   1000.6;
      AN    M      3.3;
      O     ;
      A     M   1000.5;
      A     DB51.DBX  208.1;
      A     DB51.DBX  203.6;
      AN    DB51.DBX  203.7;
      )     ;
      A     M   1205.3;
      A     M   1204.7;
      =     L      0.0;
      A     L      0.0;
      AN    M   1202.2;
      AN    M   1240.3;
      =     M   1240.2;
      A     L      0.0;
      AN    M   1202.4;
      AN    M   1240.5;
      =     M   1240.4;
NETWORK
TITLE =

      A(    ;
      A     M   1000.6;
      AN    M      3.3;
      O     ;
      A     M   1000.5;
      A     DB51.DBX  208.1;
      A     DB51.DBX  203.7;
      AN    DB51.DBX  203.6;
      O     M   1001.2;
      )     ;
      A     M   1205.3;
      A     M   1204.7;
      =     L      0.0;
      A     L      0.0;
      AN    M   1202.3;
      AN    M   1240.2;
      =     M   1240.3;
      A     L      0.0;
      AN    M   1202.5;
      AN    M   1240.4;
      =     M   1240.5;
NETWORK
TITLE =

      A(    ;
      A     M   1000.6;
      AN    M      3.3;
      O     ;
      A     M   1000.5;
      A     DB51.DBX  208.2;
      A     DB51.DBX  203.6;
      AN    DB51.DBX  203.7;
      )     ;
      A     M   1205.0;
      =     L      0.0;
      A     L      0.0;
      AN    M   1202.6;
      AN    M   1240.7;
      =     M   1240.6;
      A     L      0.0;
      AN    M   1203.0;
      AN    M   1241.1;
      =     M   1241.0;
      A     L      0.0;
      AN    M   1203.2;
      AN    M   1241.3;
      =     M   1241.2;
NETWORK
TITLE =
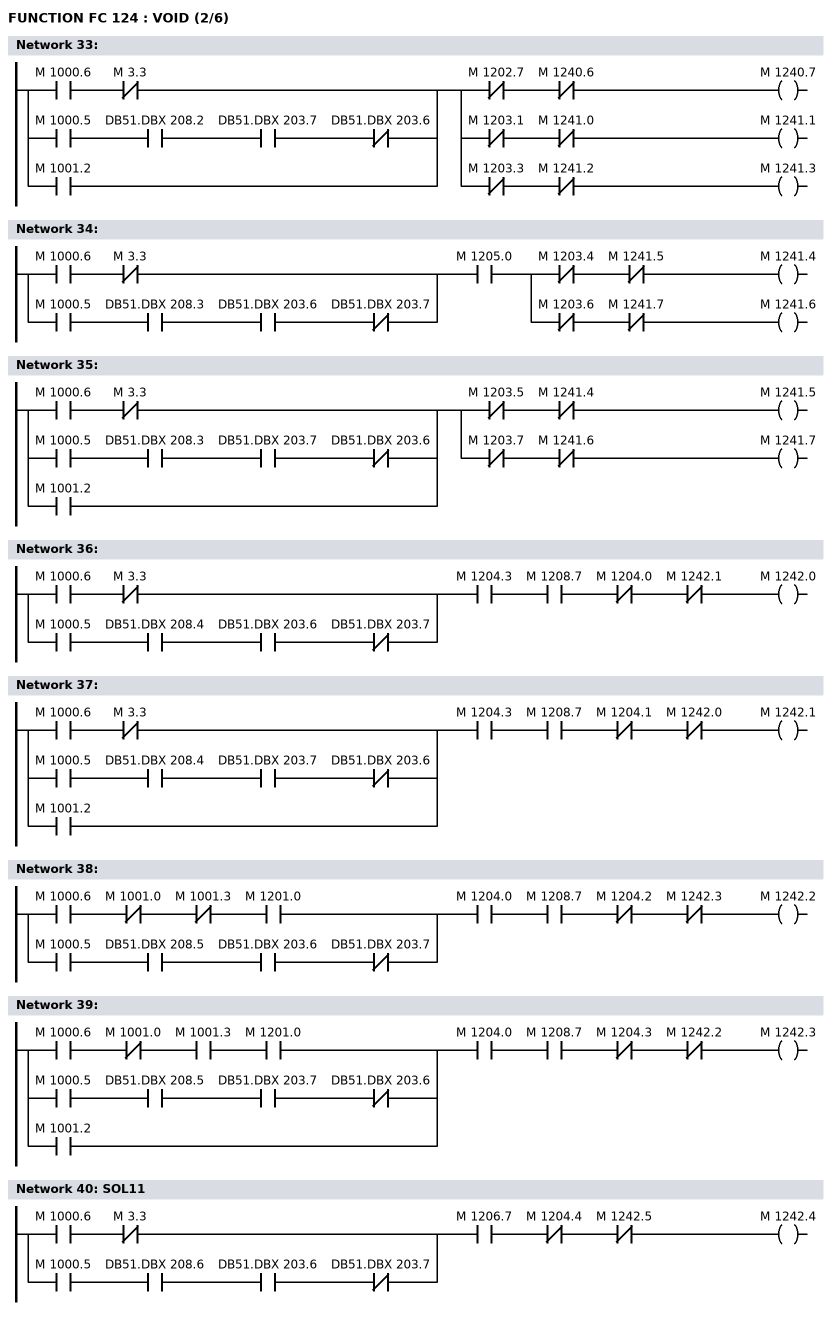

      A     M   1000.6;
      AN    M      3.3;
      O     ;
      A     M   1000.5;
      A     DB51.DBX  208.2;
      A     DB51.DBX  203.7;
      AN    DB51.DBX  203.6;
      O     M   1001.2;
      =     L      0.0;
      A     L      0.0;
      AN    M   1202.7;
      AN    M   1240.6;
      =     M   1240.7;
      A     L      0.0;
      AN    M   1203.1;
      AN    M   1241.0;
      =     M   1241.1;
      A     L      0.0;
      AN    M   1203.3;
      AN    M   1241.2;
      =     M   1241.3;
NETWORK
TITLE =

      A(    ;
      A     M   1000.6;
      AN    M      3.3;
      O     ;
      A     M   1000.5;
      A     DB51.DBX  208.3;
      A     DB51.DBX  203.6;
      AN    DB51.DBX  203.7;
      )     ;
      A     M   1205.0;
      =     L      0.0;
      A     L      0.0;
      AN    M   1203.4;
      AN    M   1241.5;
      =     M   1241.4;
      A     L      0.0;
      AN    M   1203.6;
      AN    M   1241.7;
      =     M   1241.6;
NETWORK
TITLE =

      A     M   1000.6;
      AN    M      3.3;
      O     ;
      A     M   1000.5;
      A     DB51.DBX  208.3;
      A     DB51.DBX  203.7;
      AN    DB51.DBX  203.6;
      O     M   1001.2;
      =     L      0.0;
      A     L      0.0;
      AN    M   1203.5;
      AN    M   1241.4;
      =     M   1241.5;
      A     L      0.0;
      AN    M   1203.7;
      AN    M   1241.6;
      =     M   1241.7;
NETWORK
TITLE =

      A(    ;
      A     M   1000.6;
      AN    M      3.3;
      O     ;
      A     M   1000.5;
      A     DB51.DBX  208.4;
      A     DB51.DBX  203.6;
      AN    DB51.DBX  203.7;
      )     ;
      A     M   1204.3;
      A     M   1208.7;
      AN    M   1204.0;
      AN    M   1242.1;
      =     M   1242.0;
NETWORK
TITLE =

      A(    ;
      A     M   1000.6;
      AN    M      3.3;
      O     ;
      A     M   1000.5;
      A     DB51.DBX  208.4;
      A     DB51.DBX  203.7;
      AN    DB51.DBX  203.6;
      O     M   1001.2;
      )     ;
      A     M   1204.3;
      A     M   1208.7;
      AN    M   1204.1;
      AN    M   1242.0;
      =     M   1242.1;
NETWORK
TITLE =

      A(    ;
      A     M   1000.6;
      AN    M   1001.0;
      AN    M   1001.3;
      A     M   1201.0;
      O     ;
      A     M   1000.5;
      A     DB51.DBX  208.5;
      A     DB51.DBX  203.6;
      AN    DB51.DBX  203.7;
      )     ;
      A     M   1204.0;
      A     M   1208.7;
      AN    M   1204.2;
      AN    M   1242.3;
      =     M   1242.2;
NETWORK
TITLE =

      A(    ;
      A     M   1000.6;
      AN    M   1001.0;
      A     M   1001.3;
      A     M   1201.0;
      O     ;
      A     M   1000.5;
      A     DB51.DBX  208.5;
      A     DB51.DBX  203.7;
      AN    DB51.DBX  203.6;
      O     M   1001.2;
      )     ;
      A     M   1204.0;
      A     M   1208.7;
      AN    M   1204.3;
      AN    M   1242.2;
      =     M   1242.3;
NETWORK
TITLE =SOL11

      A(    ;
      A     M   1000.6;
      AN    M      3.3;
      O     ;
      A     M   1000.5;
      A     DB51.DBX  208.6;
      A     DB51.DBX  203.6;
      AN    DB51.DBX  203.7;
      )     ;
      A     M   1206.7;
      AN    M   1204.4;
      AN    M   1242.5;
      =     M   1242.4;
NETWORK
TITLE =
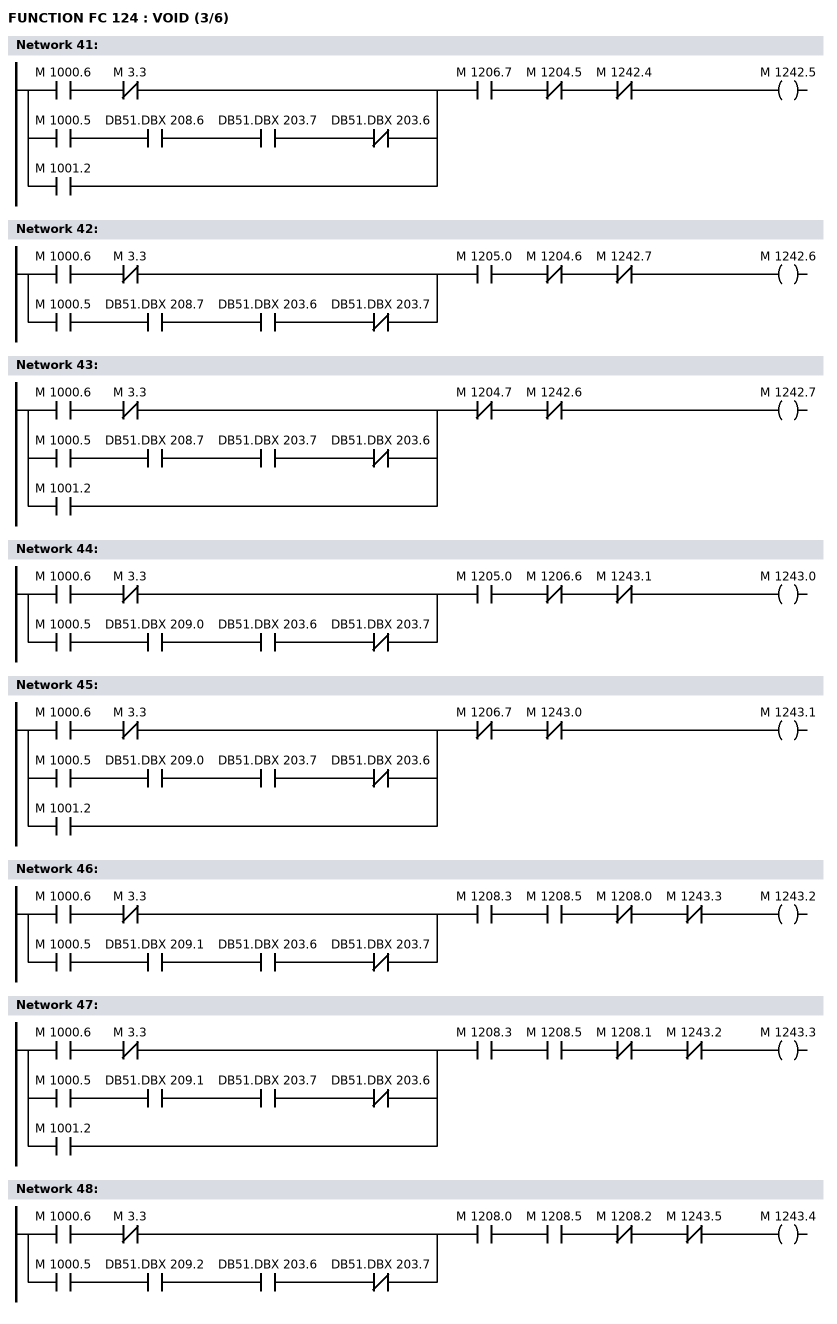

      A(    ;
      A     M   1000.6;
      AN    M      3.3;
      O     ;
      A     M   1000.5;
      A     DB51.DBX  208.6;
      A     DB51.DBX  203.7;
      AN    DB51.DBX  203.6;
      O     M   1001.2;
      )     ;
      A     M   1206.7;
      AN    M   1204.5;
      AN    M   1242.4;
      =     M   1242.5;
NETWORK
TITLE =

      A(    ;
      A     M   1000.6;
      AN    M      3.3;
      O     ;
      A     M   1000.5;
      A     DB51.DBX  208.7;
      A     DB51.DBX  203.6;
      AN    DB51.DBX  203.7;
      )     ;
      A     M   1205.0;
      AN    M   1204.6;
      AN    M   1242.7;
      =     M   1242.6;
NETWORK
TITLE =

      A(    ;
      A     M   1000.6;
      AN    M      3.3;
      O     ;
      A     M   1000.5;
      A     DB51.DBX  208.7;
      A     DB51.DBX  203.7;
      AN    DB51.DBX  203.6;
      O     M   1001.2;
      )     ;
      AN    M   1204.7;
      AN    M   1242.6;
      =     M   1242.7;
NETWORK
TITLE =

      A(    ;
      A     M   1000.6;
      AN    M      3.3;
      O     ;
      A     M   1000.5;
      A     DB51.DBX  209.0;
      A     DB51.DBX  203.6;
      AN    DB51.DBX  203.7;
      )     ;
      A     M   1205.0;
      AN    M   1206.6;
      AN    M   1243.1;
      =     M   1243.0;
NETWORK
TITLE =

      A(    ;
      A     M   1000.6;
      AN    M      3.3;
      O     ;
      A     M   1000.5;
      A     DB51.DBX  209.0;
      A     DB51.DBX  203.7;
      AN    DB51.DBX  203.6;
      O     M   1001.2;
      )     ;
      AN    M   1206.7;
      AN    M   1243.0;
      =     M   1243.1;
NETWORK
TITLE =

      A(    ;
      A     M   1000.6;
      AN    M      3.3;
      O     ;
      A     M   1000.5;
      A     DB51.DBX  209.1;
      A     DB51.DBX  203.6;
      AN    DB51.DBX  203.7;
      )     ;
      A     M   1208.3;
      A     M   1208.5;
      AN    M   1208.0;
      AN    M   1243.3;
      =     M   1243.2;
NETWORK
TITLE =

      A(    ;
      A     M   1000.6;
      AN    M      3.3;
      O     ;
      A     M   1000.5;
      A     DB51.DBX  209.1;
      A     DB51.DBX  203.7;
      AN    DB51.DBX  203.6;
      O     M   1001.2;
      )     ;
      A     M   1208.3;
      A     M   1208.5;
      AN    M   1208.1;
      AN    M   1243.2;
      =     M   1243.3;
NETWORK
TITLE =

      A(    ;
      A     M   1000.6;
      AN    M      3.3;
      O     ;
      A     M   1000.5;
      A     DB51.DBX  209.2;
      A     DB51.DBX  203.6;
      AN    DB51.DBX  203.7;
      )     ;
      A     M   1208.0;
      A     M   1208.5;
      AN    M   1208.2;
      AN    M   1243.5;
      =     M   1243.4;
NETWORK
TITLE =
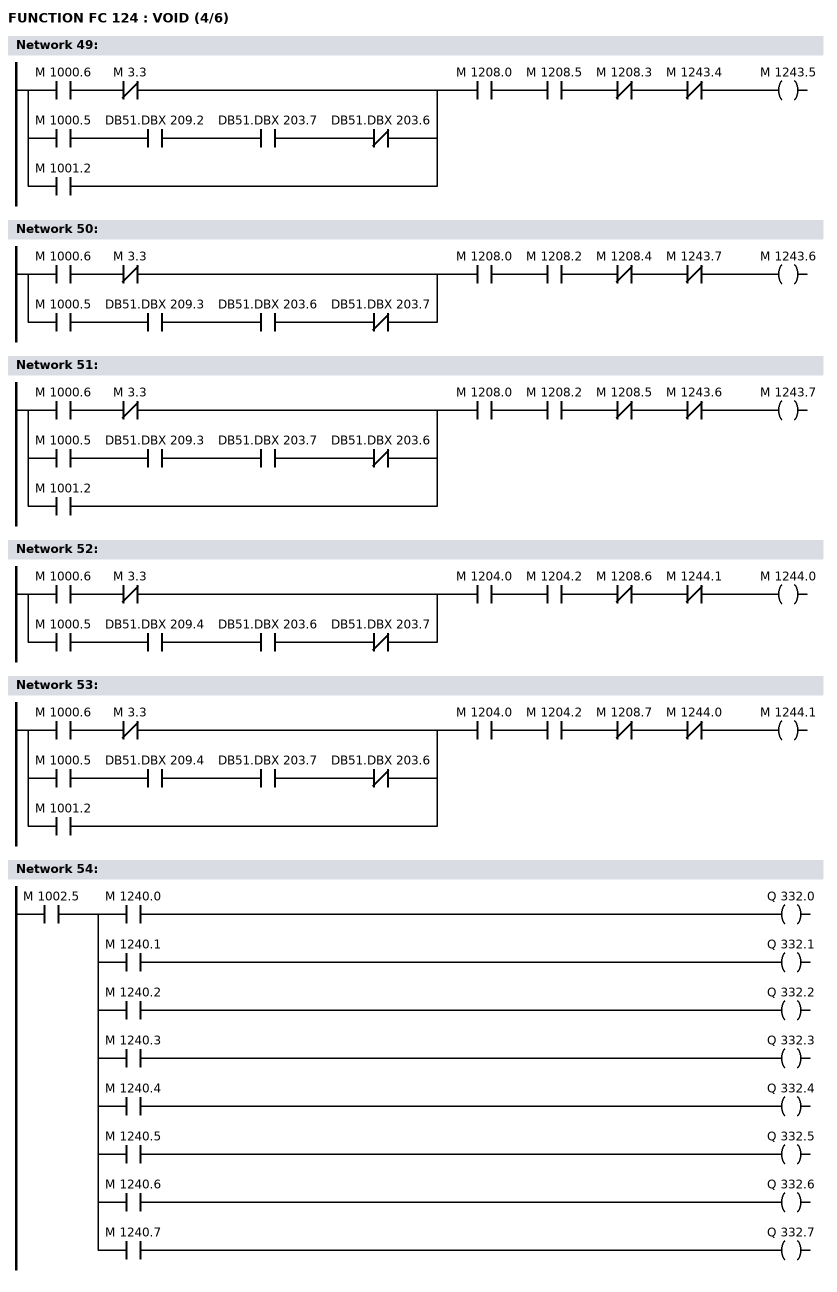

      A(    ;
      A     M   1000.6;
      AN    M      3.3;
      O     ;
      A     M   1000.5;
      A     DB51.DBX  209.2;
      A     DB51.DBX  203.7;
      AN    DB51.DBX  203.6;
      O     M   1001.2;
      )     ;
      A     M   1208.0;
      A     M   1208.5;
      AN    M   1208.3;
      AN    M   1243.4;
      =     M   1243.5;
NETWORK
TITLE =

      A(    ;
      A     M   1000.6;
      AN    M      3.3;
      O     ;
      A     M   1000.5;
      A     DB51.DBX  209.3;
      A     DB51.DBX  203.6;
      AN    DB51.DBX  203.7;
      )     ;
      A     M   1208.0;
      A     M   1208.2;
      AN    M   1208.4;
      AN    M   1243.7;
      =     M   1243.6;
NETWORK
TITLE =

      A(    ;
      A     M   1000.6;
      AN    M      3.3;
      O     ;
      A     M   1000.5;
      A     DB51.DBX  209.3;
      A     DB51.DBX  203.7;
      AN    DB51.DBX  203.6;
      O     M   1001.2;
      )     ;
      A     M   1208.0;
      A     M   1208.2;
      AN    M   1208.5;
      AN    M   1243.6;
      =     M   1243.7;
NETWORK
TITLE =

      A(    ;
      A     M   1000.6;
      AN    M      3.3;
      O     ;
      A     M   1000.5;
      A     DB51.DBX  209.4;
      A     DB51.DBX  203.6;
      AN    DB51.DBX  203.7;
      )     ;
      A     M   1204.0;
      A     M   1204.2;
      AN    M   1208.6;
      AN    M   1244.1;
      =     M   1244.0;
NETWORK
TITLE =

      A(    ;
      A     M   1000.6;
      AN    M      3.3;
      O     ;
      A     M   1000.5;
      A     DB51.DBX  209.4;
      A     DB51.DBX  203.7;
      AN    DB51.DBX  203.6;
      O     M   1001.2;
      )     ;
      A     M   1204.0;
      A     M   1204.2;
      AN    M   1208.7;
      AN    M   1244.0;
      =     M   1244.1;
NETWORK
TITLE =

      A     M   1002.5;
      =     L      0.0;
      A     L      0.0;
      A     M   1240.0;
      =     Q    332.0;
      A     L      0.0;
      A     M   1240.1;
      =     Q    332.1;
      A     L      0.0;
      A     M   1240.2;
      =     Q    332.2;
      A     L      0.0;
      A     M   1240.3;
      =     Q    332.3;
      A     L      0.0;
      A     M   1240.4;
      =     Q    332.4;
      A     L      0.0;
      A     M   1240.5;
      =     Q    332.5;
      A     L      0.0;
      A     M   1240.6;
      =     Q    332.6;
      A     L      0.0;
      A     M   1240.7;
      =     Q    332.7;
NETWORK
TITLE =TL 대차 SOL 동작회로
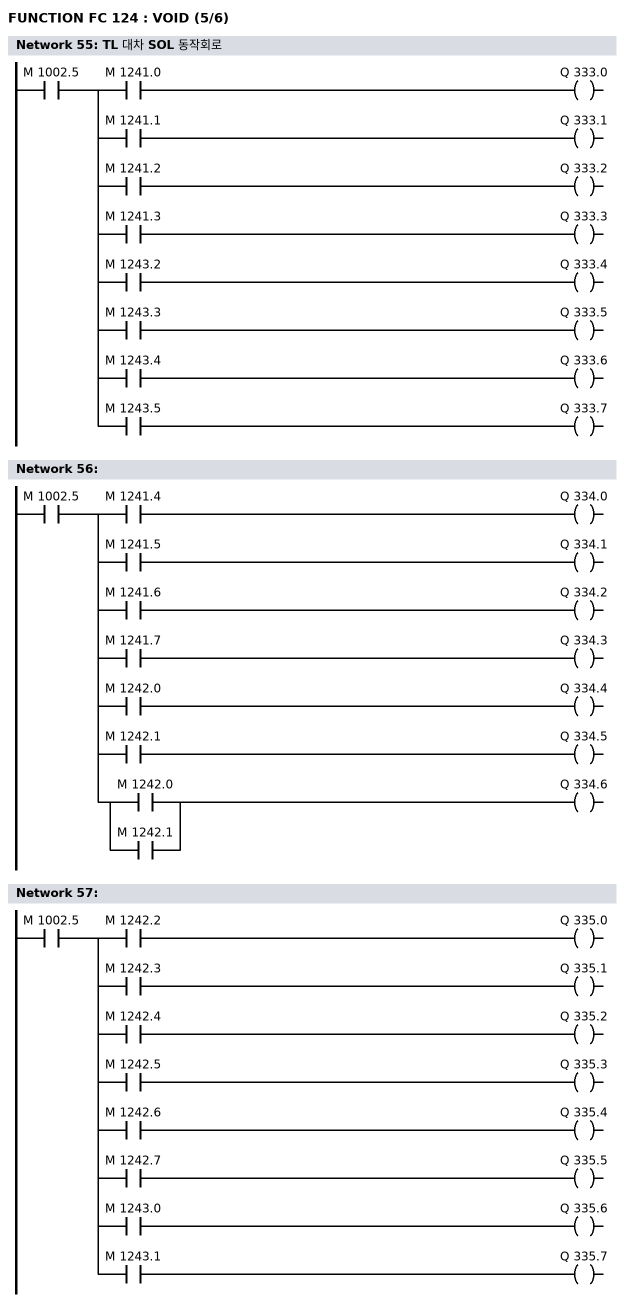

      A     M   1002.5;
      =     L      0.0;
      A     L      0.0;
      A     M   1241.0;
      =     Q    333.0;
      A     L      0.0;
      A     M   1241.1;
      =     Q    333.1;
      A     L      0.0;
      A     M   1241.2;
      =     Q    333.2;
      A     L      0.0;
      A     M   1241.3;
      =     Q    333.3;
      A     L      0.0;
      A     M   1243.2;
      =     Q    333.4;
      A     L      0.0;
      A     M   1243.3;
      =     Q    333.5;
      A     L      0.0;
      A     M   1243.4;
      =     Q    333.6;
      A     L      0.0;
      A     M   1243.5;
      =     Q    333.7;
NETWORK
TITLE =

      A     M   1002.5;
      =     L      0.0;
      A     L      0.0;
      A     M   1241.4;
      =     Q    334.0;
      A     L      0.0;
      A     M   1241.5;
      =     Q    334.1;
      A     L      0.0;
      A     M   1241.6;
      =     Q    334.2;
      A     L      0.0;
      A     M   1241.7;
      =     Q    334.3;
      A     L      0.0;
      A     M   1242.0;
      =     Q    334.4;
      A     L      0.0;
      A     M   1242.1;
      =     Q    334.5;
      A     L      0.0;
      A(    ;
      O     M   1242.0;
      O     M   1242.1;
      )     ;
      =     Q    334.6;
NETWORK
TITLE =

      A     M   1002.5;
      =     L      0.0;
      A     L      0.0;
      A     M   1242.2;
      =     Q    335.0;
      A     L      0.0;
      A     M   1242.3;
      =     Q    335.1;
      A     L      0.0;
      A     M   1242.4;
      =     Q    335.2;
      A     L      0.0;
      A     M   1242.5;
      =     Q    335.3;
      A     L      0.0;
      A     M   1242.6;
      =     Q    335.4;
      A     L      0.0;
      A     M   1242.7;
      =     Q    335.5;
      A     L      0.0;
      A     M   1243.0;
      =     Q    335.6;
      A     L      0.0;
      A     M   1243.1;
      =     Q    335.7;
NETWORK
TITLE =
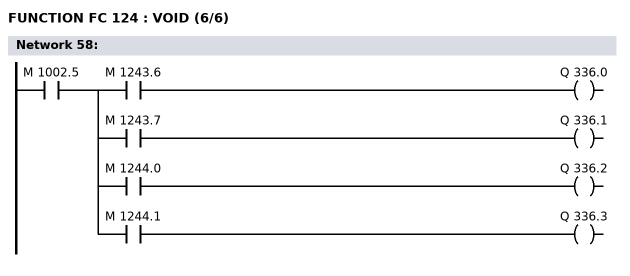

      A     M   1002.5;
      =     L      0.0;
      A     L      0.0;
      A     M   1243.6;
      =     Q    336.0;
      A     L      0.0;
      A     M   1243.7;
      =     Q    336.1;
      A     L      0.0;
      A     M   1244.0;
      =     Q    336.2;
      A     L      0.0;
      A     M   1244.1;
      =     Q    336.3;
END_FUNCTION

FUNCTION FC 125 : VOID
TITLE =
VERSION : 0.1

BEGIN
NETWORK
TITLE =
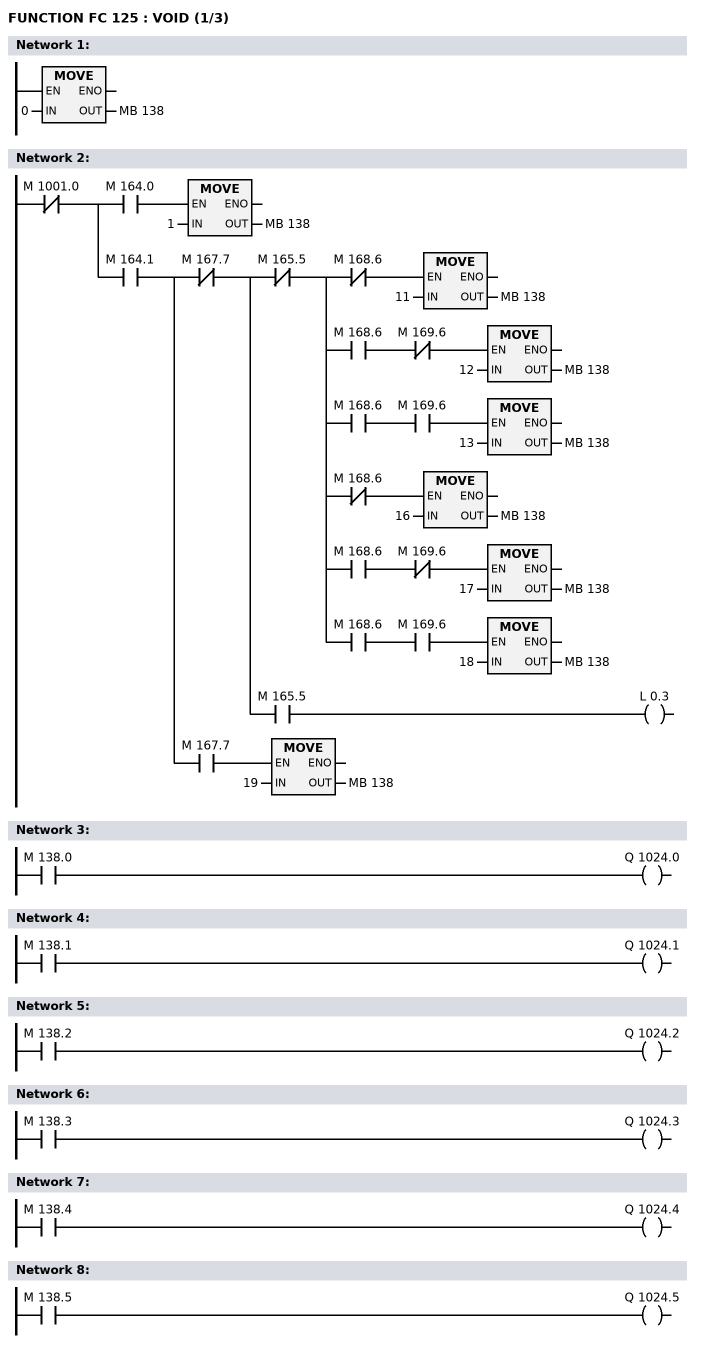

      L     0;
      T     MB   138;
      NOP   0;
NETWORK
TITLE =

      AN    M   1001.0;
      =     L      0.0;
      A     L      0.0;
      A     M    164.0;
      JNB   M001;
      L     1;
      T     MB   138;
M001: NOP   0;
      A     L      0.0;
      A     M    164.1;
      =     L      0.1;
      A     L      0.1;
      AN    M    167.7;
      =     L      0.2;
      A     L      0.2;
      AN    M    165.5;
      =     L      0.3;
      A     L      0.3;
      AN    M    168.6;
      JNB   M002;
      L     11;
      T     MB   138;
M002: NOP   0;
      A     L      0.3;
      A     M    168.6;
      AN    M    169.6;
      JNB   M003;
      L     12;
      T     MB   138;
M003: NOP   0;
      A     L      0.3;
      A     M    168.6;
      A     M    169.6;
      JNB   M004;
      L     13;
      T     MB   138;
M004: NOP   0;
      A     L      0.2;
      A     M    165.5;
      =     L      0.3;
      A     L      0.3;
      AN    M    168.6;
      JNB   M005;
      L     16;
      T     MB   138;
M005: NOP   0;
      A     L      0.3;
      A     M    168.6;
      AN    M    169.6;
      JNB   M006;
      L     17;
      T     MB   138;
M006: NOP   0;
      A     L      0.3;
      A     M    168.6;
      A     M    169.6;
      JNB   M007;
      L     18;
      T     MB   138;
M007: NOP   0;
      A     L      0.1;
      A     M    167.7;
      JNB   M008;
      L     19;
      T     MB   138;
M008: NOP   0;
NETWORK
TITLE =

      A     M    138.0;
      =     Q   1024.0;
NETWORK
TITLE =

      A     M    138.1;
      =     Q   1024.1;
NETWORK
TITLE =

      A     M    138.2;
      =     Q   1024.2;
NETWORK
TITLE =

      A     M    138.3;
      =     Q   1024.3;
NETWORK
TITLE =

      A     M    138.4;
      =     Q   1024.4;
NETWORK
TITLE =

      A     M    138.5;
      =     Q   1024.5;
NETWORK
TITLE =
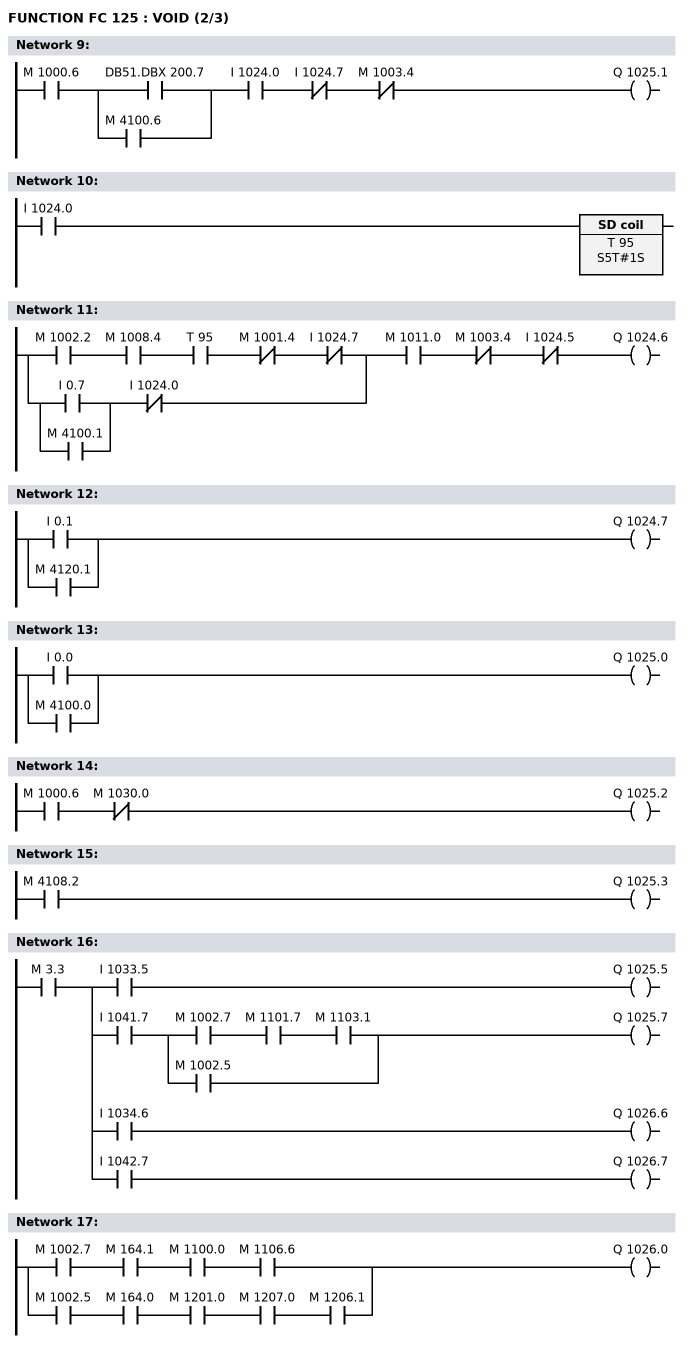

      A     M   1000.6;
      A(    ;
      O     DB51.DBX  200.7;
      O     M   4100.6;
      )     ;
      A     I   1024.0;
      AN    I   1024.7;
      AN    M   1003.4;
      =     Q   1025.1;
NETWORK
TITLE =

      A     I   1024.0;
      L     S5T#1S;
      SD    T     95;
NETWORK
TITLE =

      A(    ;
      A     M   1002.2;
      A     M   1008.4;
      A     T     95;
      AN    M   1001.4;
      AN    I   1024.7;
      O     ;
      A(    ;
      O     I      0.7;
      O     M   4100.1;
      )     ;
      AN    I   1024.0;
      )     ;
      A     M   1011.0;
      AN    M   1003.4;
      AN    I   1024.5;
      =     Q   1024.6;
NETWORK
TITLE =

      O     I      0.1;
      O     M   4120.1;
      =     Q   1024.7;
NETWORK
TITLE =

      O     I      0.0;
      O     M   4100.0;
      =     Q   1025.0;
NETWORK
TITLE =

      A     M   1000.6;
      AN    M   1030.0;
      =     Q   1025.2;
NETWORK
TITLE =

      A     M   4108.2;
      =     Q   1025.3;
NETWORK
TITLE =

      A     M      3.3;
      =     L      0.0;
      A     L      0.0;
      A     I   1033.5;
      =     Q   1025.5;
      A     L      0.0;
      A     I   1041.7;
      A(    ;
      A     M   1002.7;
      A     M   1101.7;
      A     M   1103.1;
      O     M   1002.5;
      )     ;
      =     Q   1025.7;
      A     L      0.0;
      A     I   1034.6;
      =     Q   1026.6;
      A     L      0.0;
      A     I   1042.7;
      =     Q   1026.7;
NETWORK
TITLE =

      A     M   1002.7;
      A     M    164.1;
      A     M   1100.0;
      A     M   1106.6;
      O     ;
      A     M   1002.5;
      A     M    164.0;
      A     M   1201.0;
      A     M   1207.0;
      A     M   1206.1;
      =     Q   1026.0;
NETWORK
TITLE =
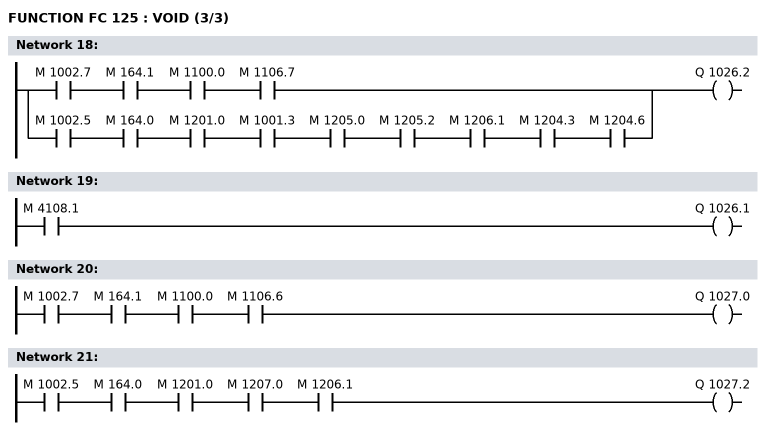

      A     M   1002.7;
      A     M    164.1;
      A     M   1100.0;
      A     M   1106.7;
      O     ;
      A     M   1002.5;
      A     M    164.0;
      A     M   1201.0;
      A     M   1001.3;
      A     M   1205.0;
      A     M   1205.2;
      A     M   1206.1;
      A     M   1204.3;
      A     M   1204.6;
      =     Q   1026.2;
NETWORK
TITLE =

      A     M   4108.1;
      =     Q   1026.1;
NETWORK
TITLE =

      A     M   1002.7;
      A     M    164.1;
      A     M   1100.0;
      A     M   1106.6;
      =     Q   1027.0;
NETWORK
TITLE =

      A     M   1002.5;
      A     M    164.0;
      A     M   1201.0;
      A     M   1207.0;
      A     M   1206.1;
      =     Q   1027.2;
END_FUNCTION

FUNCTION FC 126 : VOID
TITLE =
VERSION : 0.1

BEGIN
NETWORK
TITLE =
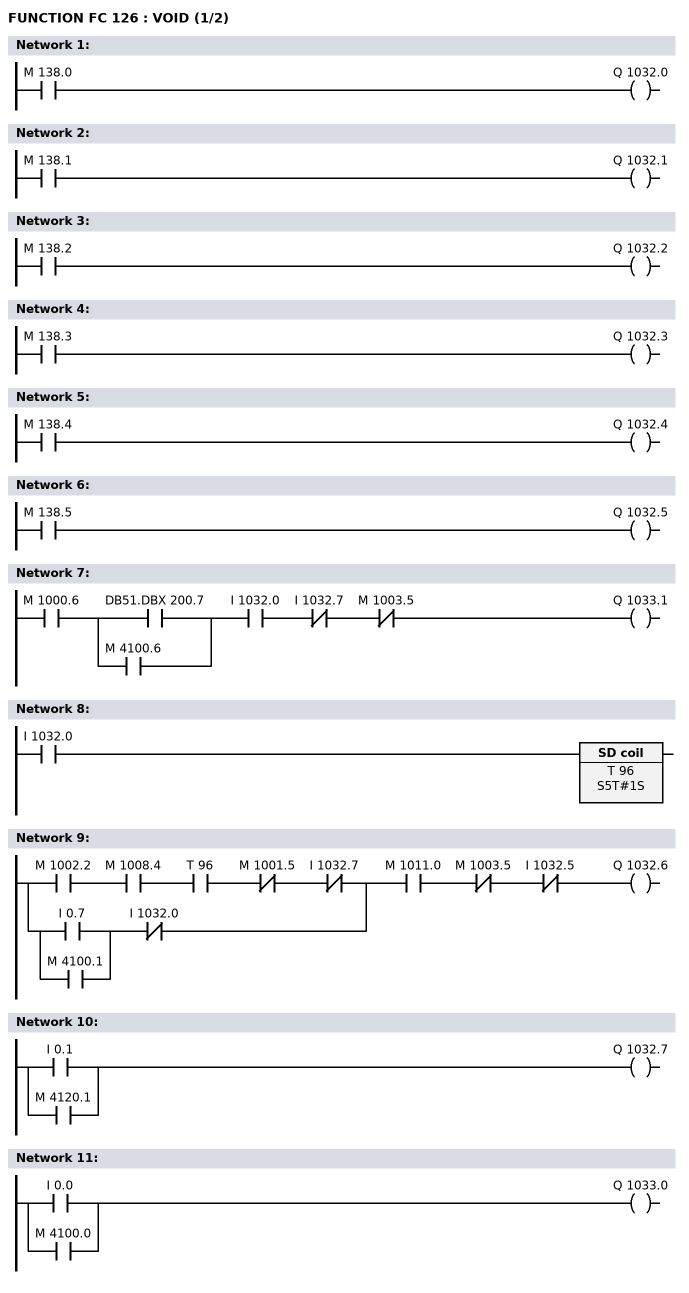

      A     M    138.0;
      =     Q   1032.0;
NETWORK
TITLE =

      A     M    138.1;
      =     Q   1032.1;
NETWORK
TITLE =

      A     M    138.2;
      =     Q   1032.2;
NETWORK
TITLE =

      A     M    138.3;
      =     Q   1032.3;
NETWORK
TITLE =

      A     M    138.4;
      =     Q   1032.4;
NETWORK
TITLE =

      A     M    138.5;
      =     Q   1032.5;
NETWORK
TITLE =

      A     M   1000.6;
      A(    ;
      O     DB51.DBX  200.7;
      O     M   4100.6;
      )     ;
      A     I   1032.0;
      AN    I   1032.7;
      AN    M   1003.5;
      =     Q   1033.1;
NETWORK
TITLE =

      A     I   1032.0;
      L     S5T#1S;
      SD    T     96;
NETWORK
TITLE =

      A(    ;
      A     M   1002.2;
      A     M   1008.4;
      A     T     96;
      AN    M   1001.5;
      AN    I   1032.7;
      O     ;
      A(    ;
      O     I      0.7;
      O     M   4100.1;
      )     ;
      AN    I   1032.0;
      )     ;
      A     M   1011.0;
      AN    M   1003.5;
      AN    I   1032.5;
      =     Q   1032.6;
NETWORK
TITLE =

      O     I      0.1;
      O     M   4120.1;
      =     Q   1032.7;
NETWORK
TITLE =

      O     I      0.0;
      O     M   4100.0;
      =     Q   1033.0;
NETWORK
TITLE =
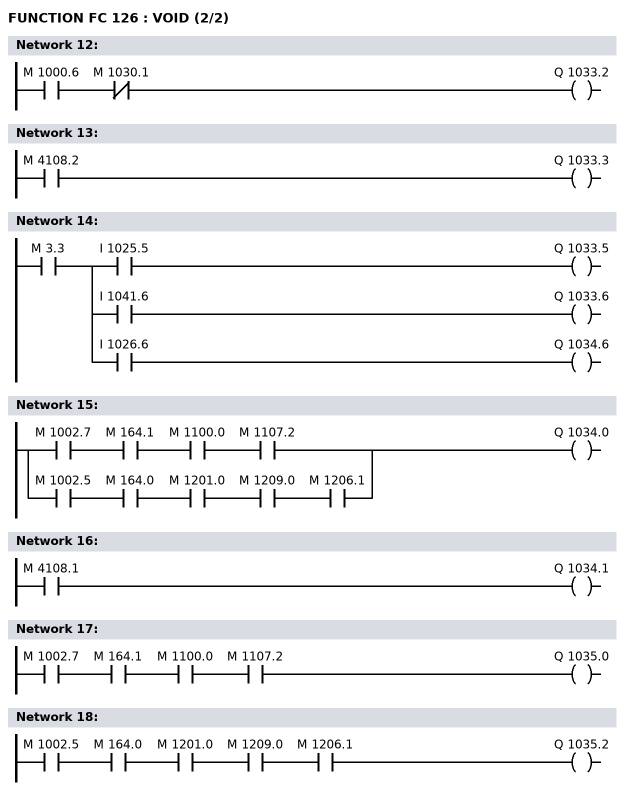

      A     M   1000.6;
      AN    M   1030.1;
      =     Q   1033.2;
NETWORK
TITLE =

      A     M   4108.2;
      =     Q   1033.3;
NETWORK
TITLE =

      A     M      3.3;
      =     L      0.0;
      A     L      0.0;
      A     I   1025.5;
      =     Q   1033.5;
      A     L      0.0;
      A     I   1041.6;
      =     Q   1033.6;
      A     L      0.0;
      A     I   1026.6;
      =     Q   1034.6;
NETWORK
TITLE =

      A     M   1002.7;
      A     M    164.1;
      A     M   1100.0;
      A     M   1107.2;
      O     ;
      A     M   1002.5;
      A     M    164.0;
      A     M   1201.0;
      A     M   1209.0;
      A     M   1206.1;
      =     Q   1034.0;
NETWORK
TITLE =

      A     M   4108.1;
      =     Q   1034.1;
NETWORK
TITLE =

      A     M   1002.7;
      A     M    164.1;
      A     M   1100.0;
      A     M   1107.2;
      =     Q   1035.0;
NETWORK
TITLE =

      A     M   1002.5;
      A     M    164.0;
      A     M   1201.0;
      A     M   1209.0;
      A     M   1206.1;
      =     Q   1035.2;
END_FUNCTION

FUNCTION FC 127 : VOID
TITLE =
VERSION : 0.1

BEGIN
NETWORK
TITLE =
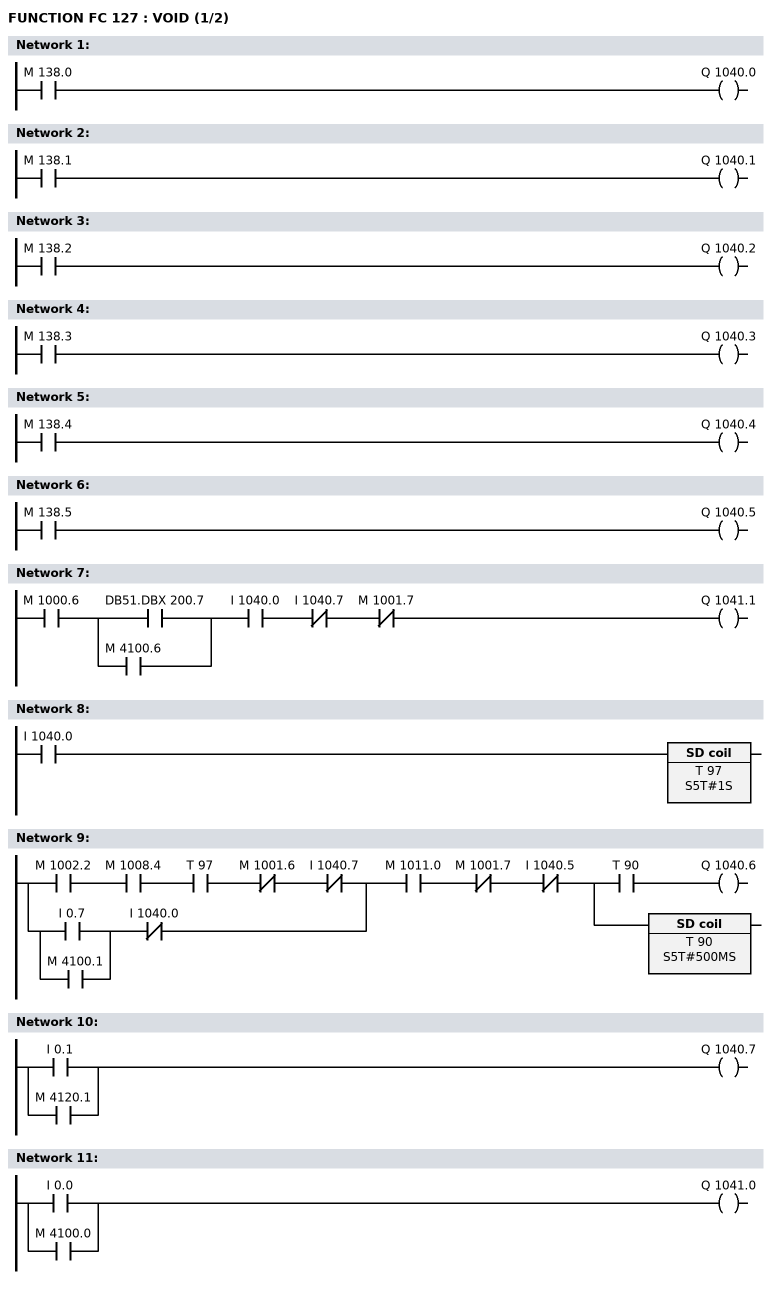

      A     M    138.0;
      =     Q   1040.0;
NETWORK
TITLE =

      A     M    138.1;
      =     Q   1040.1;
NETWORK
TITLE =

      A     M    138.2;
      =     Q   1040.2;
NETWORK
TITLE =

      A     M    138.3;
      =     Q   1040.3;
NETWORK
TITLE =

      A     M    138.4;
      =     Q   1040.4;
NETWORK
TITLE =

      A     M    138.5;
      =     Q   1040.5;
NETWORK
TITLE =

      A     M   1000.6;
      A(    ;
      O     DB51.DBX  200.7;
      O     M   4100.6;
      )     ;
      A     I   1040.0;
      AN    I   1040.7;
      AN    M   1001.7;
      =     Q   1041.1;
NETWORK
TITLE =

      A     I   1040.0;
      L     S5T#1S;
      SD    T     97;
NETWORK
TITLE =

      A(    ;
      A     M   1002.2;
      A     M   1008.4;
      A     T     97;
      AN    M   1001.6;
      AN    I   1040.7;
      O     ;
      A(    ;
      O     I      0.7;
      O     M   4100.1;
      )     ;
      AN    I   1040.0;
      )     ;
      A     M   1011.0;
      AN    M   1001.7;
      AN    I   1040.5;
      =     L      0.0;
      A     L      0.0;
      A     T     90;
      =     Q   1040.6;
      A     L      0.0;
      BLD   102;
      L     S5T#500MS;
      SD    T     90;
NETWORK
TITLE =

      O     I      0.1;
      O     M   4120.1;
      =     Q   1040.7;
NETWORK
TITLE =

      O     I      0.0;
      O     M   4100.0;
      =     Q   1041.0;
NETWORK
TITLE =
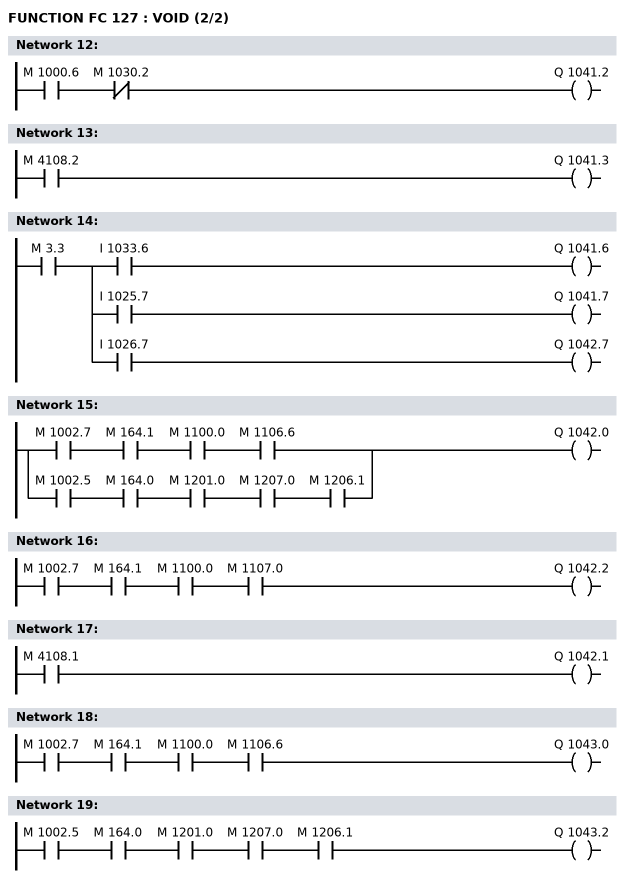

      A     M   1000.6;
      AN    M   1030.2;
      =     Q   1041.2;
NETWORK
TITLE =

      A     M   4108.2;
      =     Q   1041.3;
NETWORK
TITLE =

      A     M      3.3;
      =     L      0.0;
      A     L      0.0;
      A     I   1033.6;
      =     Q   1041.6;
      A     L      0.0;
      A     I   1025.7;
      =     Q   1041.7;
      A     L      0.0;
      A     I   1026.7;
      =     Q   1042.7;
NETWORK
TITLE =

      A     M   1002.7;
      A     M    164.1;
      A     M   1100.0;
      A     M   1106.6;
      O     ;
      A     M   1002.5;
      A     M    164.0;
      A     M   1201.0;
      A     M   1207.0;
      A     M   1206.1;
      =     Q   1042.0;
NETWORK
TITLE =

      A     M   1002.7;
      A     M    164.1;
      A     M   1100.0;
      A     M   1107.0;
      =     Q   1042.2;
NETWORK
TITLE =

      A     M   4108.1;
      =     Q   1042.1;
NETWORK
TITLE =

      A     M   1002.7;
      A     M    164.1;
      A     M   1100.0;
      A     M   1106.6;
      =     Q   1043.0;
NETWORK
TITLE =

      A     M   1002.5;
      A     M    164.0;
      A     M   1201.0;
      A     M   1207.0;
      A     M   1206.1;
      =     Q   1043.2;
END_FUNCTION

FUNCTION_BLOCK FB 130
TITLE =
VERSION : 0.1


VAR
  S707_MODE : FB 402;
END_VAR
BEGIN
NETWORK
TITLE =
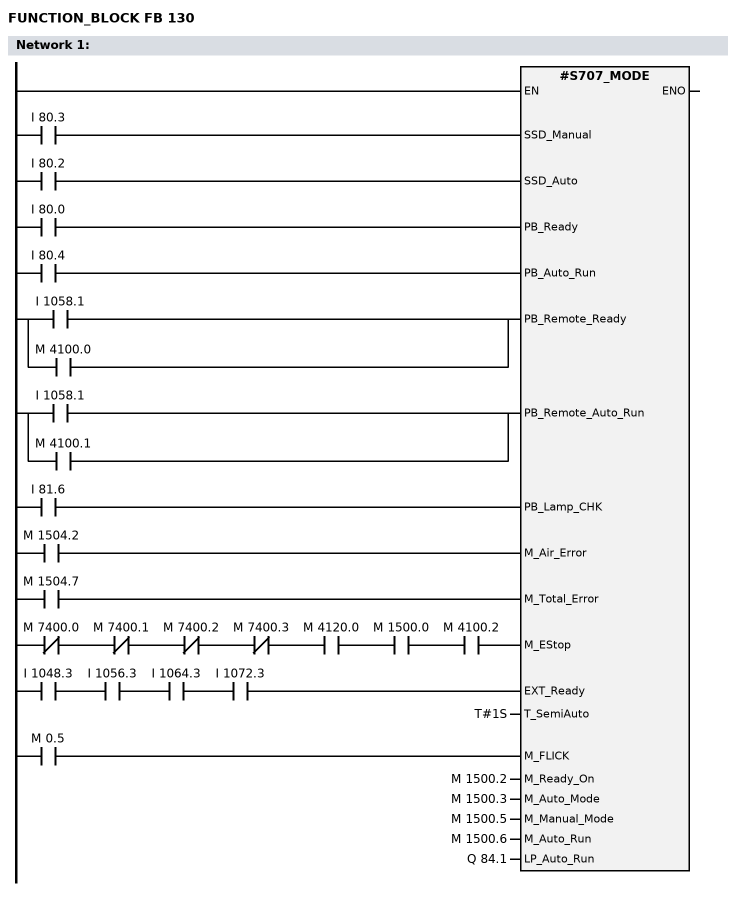

      A     I     80.3;
      =     L      0.0;
      BLD   103;
      A     I     80.2;
      =     L      0.1;
      BLD   103;
      A     I     80.0;
      =     L      0.2;
      BLD   103;
      A     I     80.4;
      =     L      0.3;
      BLD   103;
      A(    ;
      O     I   1058.1;
      O     M   4100.0;
      )     ;
      =     L      0.4;
      BLD   103;
      A(    ;
      O     I   1058.1;
      O     M   4100.1;
      )     ;
      =     L      0.5;
      BLD   103;
      A     I     81.6;
      =     L      0.6;
      BLD   103;
      A     M   1504.2;
      =     L      0.7;
      BLD   103;
      A     M   1504.7;
      =     L      1.1;
      BLD   103;
      AN    M   7400.0;
      AN    M   7400.1;
      AN    M   7400.2;
      AN    M   7400.3;
      A     M   4120.0;
      A     M   1500.0;
      A     M   4100.2;
      =     L      1.2;
      BLD   103;
      A     I   1048.3;
      A     I   1056.3;
      A     I   1064.3;
      A     I   1072.3;
      =     L      1.3;
      BLD   103;
      A     M      0.5;
      =     L      1.5;
      BLD   103;
      CALL #S707_MODE (
           SSD_Manual               := L      0.0,
           SSD_Auto                 := L      0.1,
           PB_Ready                 := L      0.2,
           PB_Auto_Run              := L      0.3,
           PB_Remote_Ready          := L      0.4,
           PB_Remote_Auto_Run       := L      0.5,
           PB_Lamp_CHK              := L      0.6,
           M_Air_Error              := L      0.7,
           M_Total_Error            := L      1.1,
           M_EStop                  := L      1.2,
           EXT_Ready                := L      1.3,
           T_SemiAuto               := T#1S,
           M_FLICK                  := L      1.5,
           M_Ready_On               := M   1500.2,
           M_Auto_Mode              := M   1500.3,
           M_Manual_Mode            := M   1500.5,
           M_Auto_Run               := M   1500.6,
           LP_Auto_Run              := Q     84.1);
      NOP   0;
END_FUNCTION_BLOCK

DATA_BLOCK DB 130
TITLE =
VERSION : 0.0

 FB 130
BEGIN
   S707_MODE.SSD_Manual := FALSE;
   S707_MODE.SSD_Auto := TRUE;
   S707_MODE.PB_Ready := FALSE;
   S707_MODE.PB_Auto_Run := FALSE;
   S707_MODE.PB_Remote_Ready := FALSE;
   S707_MODE.PB_Remote_Auto_Run := FALSE;
   S707_MODE.PB_Lamp_CHK := FALSE;
   S707_MODE.M_Air_Error := FALSE;
   S707_MODE.M_Water_Error := FALSE;
   S707_MODE.M_Total_Error := FALSE;
   S707_MODE.M_EStop := TRUE;
   S707_MODE.EXT_Ready := TRUE;
   S707_MODE.EXT_Auto := FALSE;
   S707_MODE.T_SemiAuto := T#1S;
   S707_MODE.M_FLICK := FALSE;
   S707_MODE.M_Ready_On := TRUE;
   S707_MODE.M_Auto_Mode := TRUE;
   S707_MODE.M_SemiAuto_Mode := FALSE;
   S707_MODE.M_Manual_Mode := FALSE;
   S707_MODE.M_Auto_Run := TRUE;
   S707_MODE.LP_Ready_On := TRUE;
   S707_MODE.LP_Auto_Run := TRUE;
   S707_MODE.AUTO_MODE_DELAY.IN := FALSE;
   S707_MODE.AUTO_MODE_DELAY.PT := T#0MS;
   S707_MODE.AUTO_MODE_DELAY.Q := FALSE;
   S707_MODE.AUTO_MODE_DELAY.ET := T#0MS;
   S707_MODE.AUTO_MODE_DELAY.STATE := B#16#0;
   S707_MODE.AUTO_MODE_DELAY.STIME := T#0MS;
   S707_MODE.AUTO_MODE_DELAY.ATIME := T#0MS;
   S707_MODE.SEMI_AUTO_DELAY.IN := FALSE;
   S707_MODE.SEMI_AUTO_DELAY.PT := T#1S;
   S707_MODE.SEMI_AUTO_DELAY.Q := FALSE;
   S707_MODE.SEMI_AUTO_DELAY.ET := T#0MS;
   S707_MODE.SEMI_AUTO_DELAY.STATE := B#16#0;
   S707_MODE.SEMI_AUTO_DELAY.STIME := T#20D59M41S158MS;
   S707_MODE.SEMI_AUTO_DELAY.ATIME := T#20D59M41S179MS;
   S707_MODE.MANUAL_DELAY.IN := FALSE;
   S707_MODE.MANUAL_DELAY.PT := T#0MS;
   S707_MODE.MANUAL_DELAY.Q := FALSE;
   S707_MODE.MANUAL_DELAY.ET := T#0MS;
   S707_MODE.MANUAL_DELAY.STATE := B#16#0;
   S707_MODE.MANUAL_DELAY.STIME := T#0MS;
   S707_MODE.MANUAL_DELAY.ATIME := T#0MS;
END_DATA_BLOCK

FUNCTION FC 130 : VOID
TITLE =
VERSION : 0.1

BEGIN
NETWORK
TITLE =
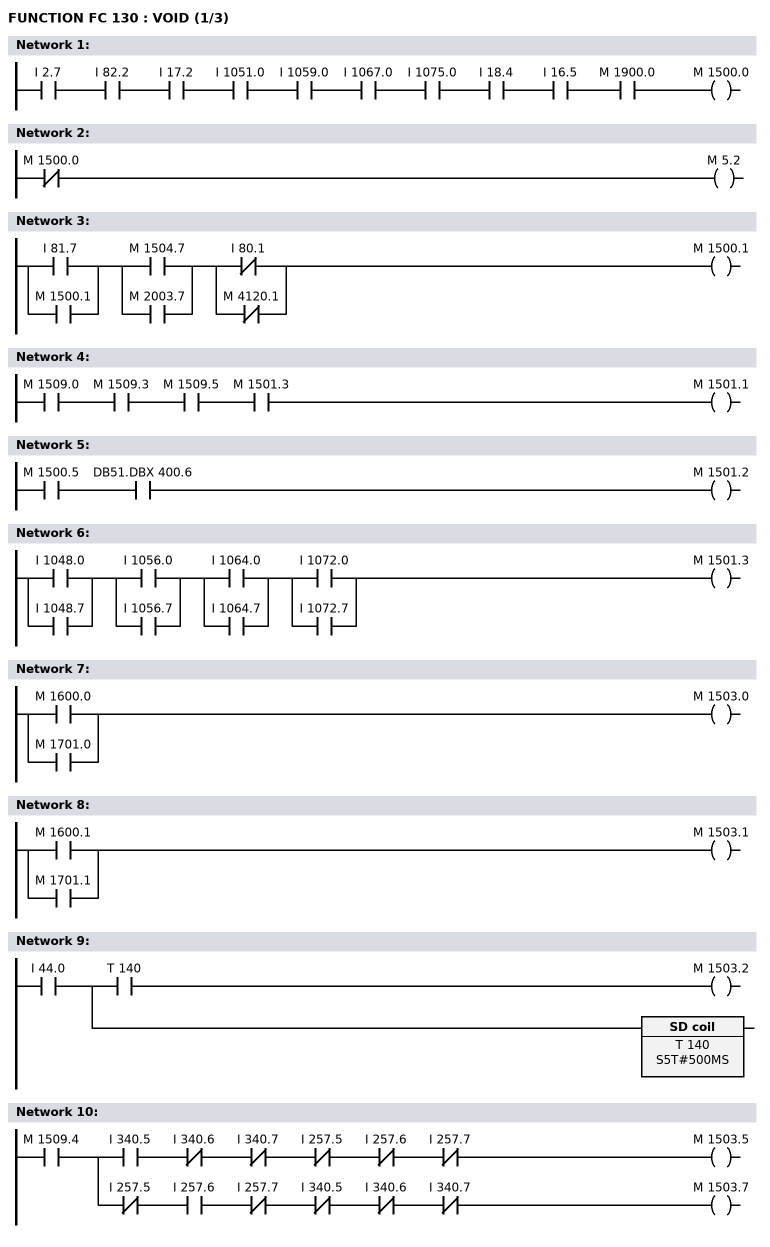

      A     I      2.7;
      A     I     82.2;
      A     I     17.2;
      A     I   1051.0;
      A     I   1059.0;
      A     I   1067.0;
      A     I   1075.0;
      A     I     18.4;
      A     I     16.5;
      A     M   1900.0;
      =     M   1500.0;
NETWORK
TITLE =

      AN    M   1500.0;
      =     M      5.2;
NETWORK
TITLE =

      A(    ;
      O     I     81.7;
      O     M   1500.1;
      )     ;
      A(    ;
      O     M   1504.7;
      O     M   2003.7;
      )     ;
      A(    ;
      ON    I     80.1;
      ON    M   4120.1;
      )     ;
      =     M   1500.1;
NETWORK
TITLE =

      A     M   1509.0;
      A     M   1509.3;
      A     M   1509.5;
      A     M   1501.3;
      =     M   1501.1;
NETWORK
TITLE =

      A     M   1500.5;
      A     DB51.DBX  400.6;
      =     M   1501.2;
NETWORK
TITLE =

      A(    ;
      O     I   1048.0;
      O     I   1048.7;
      )     ;
      A(    ;
      O     I   1056.0;
      O     I   1056.7;
      )     ;
      A(    ;
      O     I   1064.0;
      O     I   1064.7;
      )     ;
      A(    ;
      O     I   1072.0;
      O     I   1072.7;
      )     ;
      =     M   1501.3;
NETWORK
TITLE =

      O     M   1600.0;
      O     M   1701.0;
      =     M   1503.0;
NETWORK
TITLE =

      O     M   1600.1;
      O     M   1701.1;
      =     M   1503.1;
NETWORK
TITLE =

      A     I     44.0;
      =     L      0.0;
      A     L      0.0;
      A     T    140;
      =     M   1503.2;
      A     L      0.0;
      BLD   102;
      L     S5T#500MS;
      SD    T    140;
NETWORK
TITLE =

      A     M   1509.4;
      =     L      0.0;
      A     L      0.0;
      A     I    340.5;
      AN    I    340.6;
      AN    I    340.7;
      AN    I    257.5;
      AN    I    257.6;
      AN    I    257.7;
      =     M   1503.5;
      A     L      0.0;
      AN    I    257.5;
      A     I    257.6;
      AN    I    257.7;
      AN    I    340.5;
      AN    I    340.6;
      AN    I    340.7;
      =     M   1503.7;
NETWORK
TITLE =
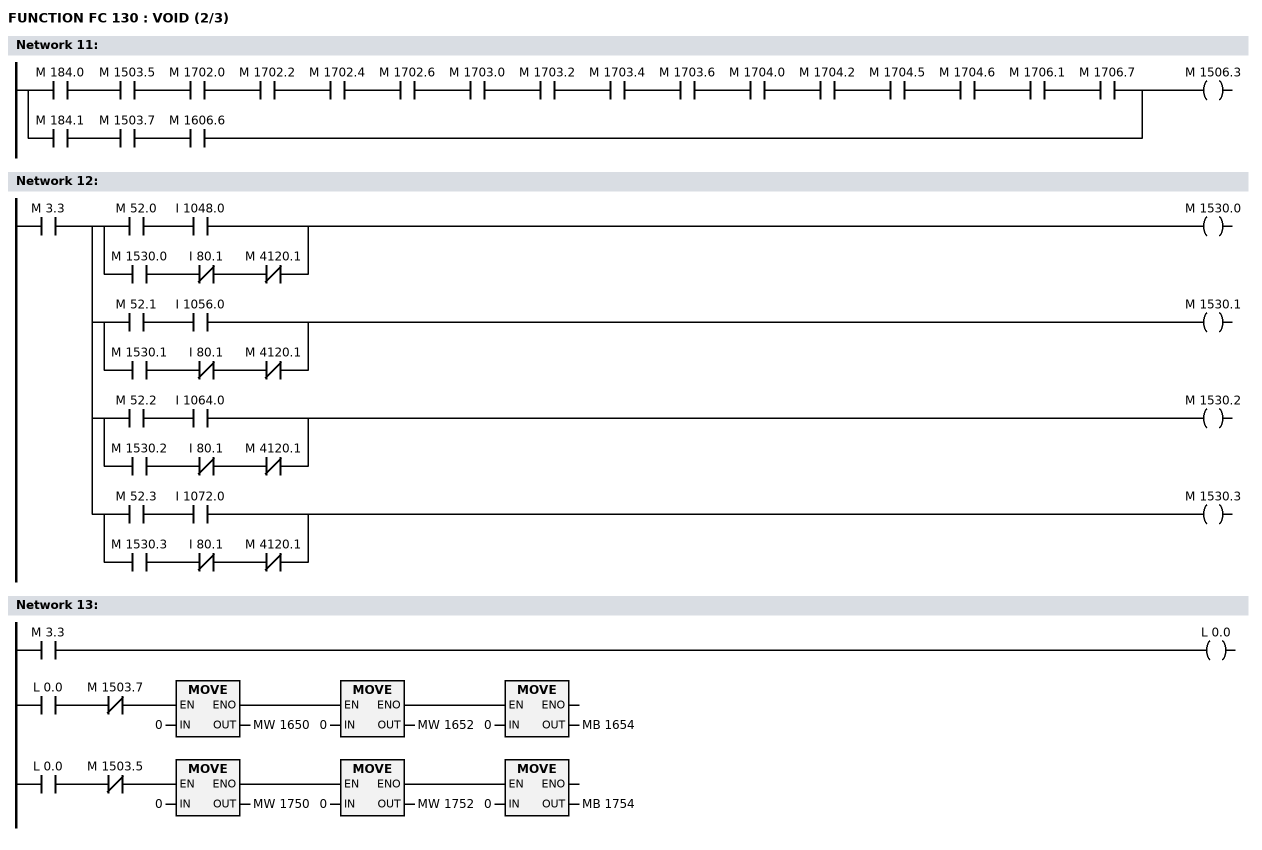

      A     M    184.0;
      A     M   1503.5;
      A     M   1702.0;
      A     M   1702.2;
      A     M   1702.4;
      A     M   1702.6;
      A     M   1703.0;
      A     M   1703.2;
      A     M   1703.4;
      A     M   1703.6;
      A     M   1704.0;
      A     M   1704.2;
      A     M   1704.5;
      A     M   1704.6;
      A     M   1706.1;
      A     M   1706.7;
      O     ;
      A     M    184.1;
      A     M   1503.7;
      A     M   1606.6;
      =     M   1506.3;
NETWORK
TITLE =

      A     M      3.3;
      =     L      0.0;
      A     L      0.0;
      A(    ;
      A     M     52.0;
      A     I   1048.0;
      O     ;
      A     M   1530.0;
      AN    I     80.1;
      AN    M   4120.1;
      )     ;
      =     M   1530.0;
      A     L      0.0;
      A(    ;
      A     M     52.1;
      A     I   1056.0;
      O     ;
      A     M   1530.1;
      AN    I     80.1;
      AN    M   4120.1;
      )     ;
      =     M   1530.1;
      A     L      0.0;
      A(    ;
      A     M     52.2;
      A     I   1064.0;
      O     ;
      A     M   1530.2;
      AN    I     80.1;
      AN    M   4120.1;
      )     ;
      =     M   1530.2;
      A     L      0.0;
      A(    ;
      A     M     52.3;
      A     I   1072.0;
      O     ;
      A     M   1530.3;
      AN    I     80.1;
      AN    M   4120.1;
      )     ;
      =     M   1530.3;
NETWORK
TITLE =

      A     M      3.3;
      =     L      0.0;
      A(    ;
      A(    ;
      A     L      0.0;
      AN    M   1503.7;
      JNB   _001;
      L     0;
      T     MW  1650;
      SET   ;
      SAVE  ;
      CLR   ;
_001: A     BR;
      )     ;
      JNB   _002;
      L     0;
      T     MW  1652;
      SET   ;
      SAVE  ;
      CLR   ;
_002: A     BR;
      )     ;
      JNB   _003;
      L     0;
      T     MB  1654;
_003: NOP   0;
      A(    ;
      A(    ;
      A     L      0.0;
      AN    M   1503.5;
      JNB   _004;
      L     0;
      T     MW  1750;
      SET   ;
      SAVE  ;
      CLR   ;
_004: A     BR;
      )     ;
      JNB   _005;
      L     0;
      T     MW  1752;
      SET   ;
      SAVE  ;
      CLR   ;
_005: A     BR;
      )     ;
      JNB   _006;
      L     0;
      T     MB  1754;
_006: NOP   0;
NETWORK
TITLE =
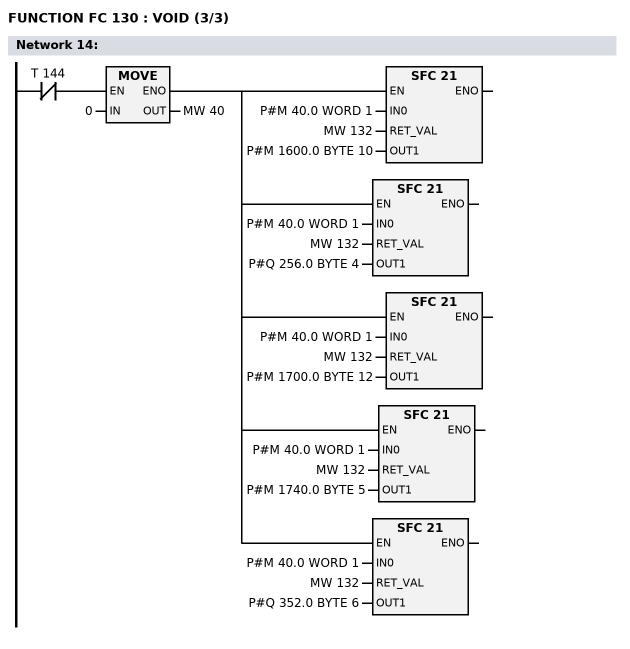

      AN    T    144;
      JNB   _007;
      L     0;
      T     MW    40;
      SET   ;
      SAVE  ;
      CLR   ;
_007: A     BR;
      =     L      0.0;
      A     L      0.0;
      JNB   _008;
      CALL SFC   21 (
           IN0                      := P#M 40.0 WORD 1,
           RET_VAL                  := MW   132,
           OUT1                     := P#M 1600.0 BYTE 10);
_008: NOP   0;
      A     L      0.0;
      JNB   _009;
      CALL SFC   21 (
           IN0                      := P#M 40.0 WORD 1,
           RET_VAL                  := MW   132,
           OUT1                     := P#Q 256.0 BYTE 4);
_009: NOP   0;
      A     L      0.0;
      JNB   _00a;
      CALL SFC   21 (
           IN0                      := P#M 40.0 WORD 1,
           RET_VAL                  := MW   132,
           OUT1                     := P#M 1700.0 BYTE 12);
_00a: NOP   0;
      A     L      0.0;
      JNB   _00b;
      CALL SFC   21 (
           IN0                      := P#M 40.0 WORD 1,
           RET_VAL                  := MW   132,
           OUT1                     := P#M 1740.0 BYTE 5);
_00b: NOP   0;
      A     L      0.0;
      JNB   _00c;
      CALL SFC   21 (
           IN0                      := P#M 40.0 WORD 1,
           RET_VAL                  := MW   132,
           OUT1                     := P#Q 352.0 BYTE 6);
_00c: NOP   0;
END_FUNCTION

FUNCTION_BLOCK FB 131
TITLE =
VERSION : 0.1


VAR
  S707_HOOK_PIN : FB 424;
  S707_DEACHA_LOCK : FB 424;
  S707_ELE : FB 424;
  S707_AIR_ELE : FB 424;
END_VAR
BEGIN
NETWORK
TITLE =
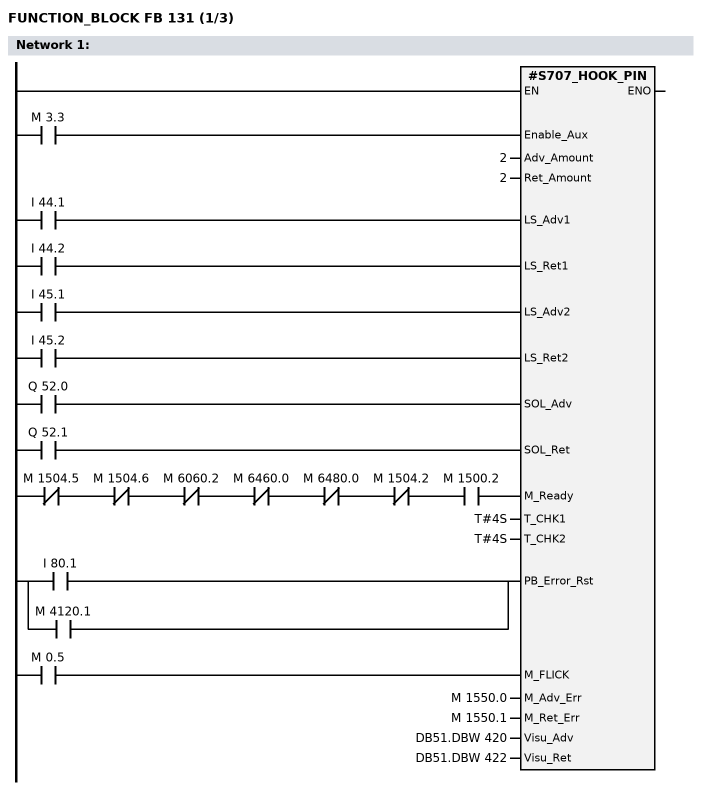

      A     M      3.3;
      =     L      0.0;
      BLD   103;
      A     I     44.1;
      =     L      0.1;
      BLD   103;
      A     I     44.2;
      =     L      0.2;
      BLD   103;
      A     I     45.1;
      =     L      0.3;
      BLD   103;
      A     I     45.2;
      =     L      0.4;
      BLD   103;
      A     Q     52.0;
      =     L      1.1;
      BLD   103;
      A     Q     52.1;
      =     L      1.2;
      BLD   103;
      AN    M   1504.5;
      AN    M   1504.6;
      AN    M   6060.2;
      AN    M   6460.0;
      AN    M   6480.0;
      AN    M   1504.2;
      A     M   1500.2;
      =     L      1.3;
      BLD   103;
      A(    ;
      O     I     80.1;
      O     M   4120.1;
      )     ;
      =     L      1.5;
      BLD   103;
      A     M      0.5;
      =     L      1.6;
      BLD   103;
      CALL #S707_HOOK_PIN (
           Enable_Aux               := L      0.0,
           Adv_Amount               := 2,
           Ret_Amount               := 2,
           LS_Adv1                  := L      0.1,
           LS_Ret1                  := L      0.2,
           LS_Adv2                  := L      0.3,
           LS_Ret2                  := L      0.4,
           SOL_Adv                  := L      1.1,
           SOL_Ret                  := L      1.2,
           M_Ready                  := L      1.3,
           T_CHK1                   := T#4S,
           T_CHK2                   := T#4S,
           PB_Error_Rst             := L      1.5,
           M_FLICK                  := L      1.6,
           M_Adv_Err                := M   1550.0,
           M_Ret_Err                := M   1550.1,
           Visu_Adv                 := DB51.DBW  420,
           Visu_Ret                 := DB51.DBW  422);
      NOP   0;
NETWORK
TITLE =
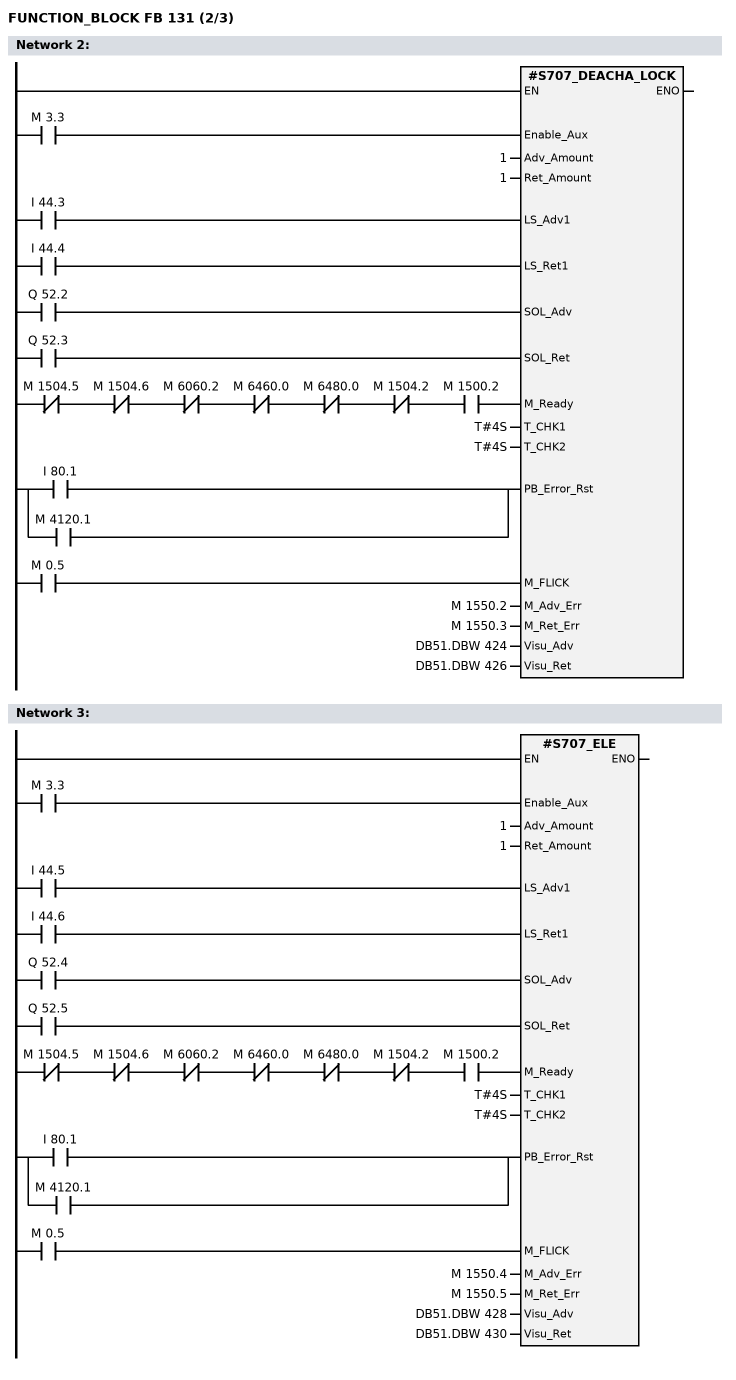

      A     M      3.3;
      =     L      0.0;
      BLD   103;
      A     I     44.3;
      =     L      0.1;
      BLD   103;
      A     I     44.4;
      =     L      0.2;
      BLD   103;
      A     Q     52.2;
      =     L      1.1;
      BLD   103;
      A     Q     52.3;
      =     L      1.2;
      BLD   103;
      AN    M   1504.5;
      AN    M   1504.6;
      AN    M   6060.2;
      AN    M   6460.0;
      AN    M   6480.0;
      AN    M   1504.2;
      A     M   1500.2;
      =     L      1.3;
      BLD   103;
      A(    ;
      O     I     80.1;
      O     M   4120.1;
      )     ;
      =     L      1.5;
      BLD   103;
      A     M      0.5;
      =     L      1.6;
      BLD   103;
      CALL #S707_DEACHA_LOCK (
           Enable_Aux               := L      0.0,
           Adv_Amount               := 1,
           Ret_Amount               := 1,
           LS_Adv1                  := L      0.1,
           LS_Ret1                  := L      0.2,
           SOL_Adv                  := L      1.1,
           SOL_Ret                  := L      1.2,
           M_Ready                  := L      1.3,
           T_CHK1                   := T#4S,
           T_CHK2                   := T#4S,
           PB_Error_Rst             := L      1.5,
           M_FLICK                  := L      1.6,
           M_Adv_Err                := M   1550.2,
           M_Ret_Err                := M   1550.3,
           Visu_Adv                 := DB51.DBW  424,
           Visu_Ret                 := DB51.DBW  426);
      NOP   0;
NETWORK
TITLE =

      A     M      3.3;
      =     L      0.0;
      BLD   103;
      A     I     44.5;
      =     L      0.1;
      BLD   103;
      A     I     44.6;
      =     L      0.2;
      BLD   103;
      A     Q     52.4;
      =     L      1.1;
      BLD   103;
      A     Q     52.5;
      =     L      1.2;
      BLD   103;
      AN    M   1504.5;
      AN    M   1504.6;
      AN    M   6060.2;
      AN    M   6460.0;
      AN    M   6480.0;
      AN    M   1504.2;
      A     M   1500.2;
      =     L      1.3;
      BLD   103;
      A(    ;
      O     I     80.1;
      O     M   4120.1;
      )     ;
      =     L      1.5;
      BLD   103;
      A     M      0.5;
      =     L      1.6;
      BLD   103;
      CALL #S707_ELE (
           Enable_Aux               := L      0.0,
           Adv_Amount               := 1,
           Ret_Amount               := 1,
           LS_Adv1                  := L      0.1,
           LS_Ret1                  := L      0.2,
           SOL_Adv                  := L      1.1,
           SOL_Ret                  := L      1.2,
           M_Ready                  := L      1.3,
           T_CHK1                   := T#4S,
           T_CHK2                   := T#4S,
           PB_Error_Rst             := L      1.5,
           M_FLICK                  := L      1.6,
           M_Adv_Err                := M   1550.4,
           M_Ret_Err                := M   1550.5,
           Visu_Adv                 := DB51.DBW  428,
           Visu_Ret                 := DB51.DBW  430);
      NOP   0;
NETWORK
TITLE =
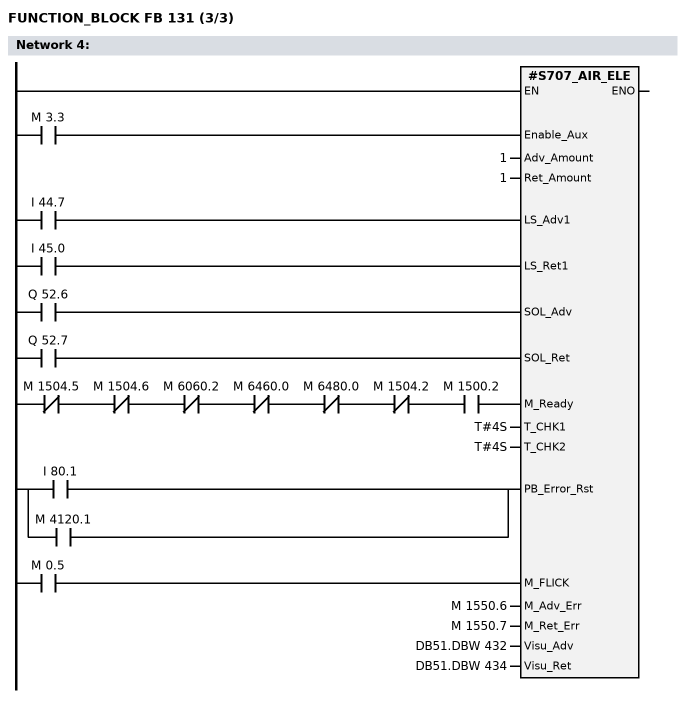

      A     M      3.3;
      =     L      0.0;
      BLD   103;
      A     I     44.7;
      =     L      0.1;
      BLD   103;
      A     I     45.0;
      =     L      0.2;
      BLD   103;
      A     Q     52.6;
      =     L      1.1;
      BLD   103;
      A     Q     52.7;
      =     L      1.2;
      BLD   103;
      AN    M   1504.5;
      AN    M   1504.6;
      AN    M   6060.2;
      AN    M   6460.0;
      AN    M   6480.0;
      AN    M   1504.2;
      A     M   1500.2;
      =     L      1.3;
      BLD   103;
      A(    ;
      O     I     80.1;
      O     M   4120.1;
      )     ;
      =     L      1.5;
      BLD   103;
      A     M      0.5;
      =     L      1.6;
      BLD   103;
      CALL #S707_AIR_ELE (
           Enable_Aux               := L      0.0,
           Adv_Amount               := 1,
           Ret_Amount               := 1,
           LS_Adv1                  := L      0.1,
           LS_Ret1                  := L      0.2,
           SOL_Adv                  := L      1.1,
           SOL_Ret                  := L      1.2,
           M_Ready                  := L      1.3,
           T_CHK1                   := T#4S,
           T_CHK2                   := T#4S,
           PB_Error_Rst             := L      1.5,
           M_FLICK                  := L      1.6,
           M_Adv_Err                := M   1550.6,
           M_Ret_Err                := M   1550.7,
           Visu_Adv                 := DB51.DBW  432,
           Visu_Ret                 := DB51.DBW  434);
      NOP   0;
END_FUNCTION_BLOCK

DATA_BLOCK DB 131
TITLE =
VERSION : 0.0

 FB 131
BEGIN
   S707_HOOK_PIN.Enable_Aux := TRUE;
   S707_HOOK_PIN.Adv_Amount := 2;
   S707_HOOK_PIN.Ret_Amount := 2;
   S707_HOOK_PIN.LS_Adv1 := FALSE;
   S707_HOOK_PIN.LS_Ret1 := TRUE;
   S707_HOOK_PIN.LS_Adv2 := FALSE;
   S707_HOOK_PIN.LS_Ret2 := TRUE;
   S707_HOOK_PIN.LS_Adv3 := FALSE;
   S707_HOOK_PIN.LS_Ret3 := FALSE;
   S707_HOOK_PIN.LS_Adv4 := FALSE;
   S707_HOOK_PIN.LS_Ret4 := FALSE;
   S707_HOOK_PIN.SOL_Adv := FALSE;
   S707_HOOK_PIN.SOL_Ret := FALSE;
   S707_HOOK_PIN.M_Ready := TRUE;
   S707_HOOK_PIN.T_CHK1 := T#4S;
   S707_HOOK_PIN.T_CHK2 := T#4S;
   S707_HOOK_PIN.PB_Lamp_CHK := FALSE;
   S707_HOOK_PIN.PB_Error_Rst := FALSE;
   S707_HOOK_PIN.M_FLICK := FALSE;
   S707_HOOK_PIN.M_Adv_Err := FALSE;
   S707_HOOK_PIN.M_Ret_Err := FALSE;
   S707_HOOK_PIN.LP_Adv := FALSE;
   S707_HOOK_PIN.LP_Ret := TRUE;
   S707_HOOK_PIN.Visu_Adv := W#16#0;
   S707_HOOK_PIN.Visu_Ret := W#16#700;
   S707_HOOK_PIN.Error_T1.IN := FALSE;
   S707_HOOK_PIN.Error_T1.PT := T#4S;
   S707_HOOK_PIN.Error_T1.Q := FALSE;
   S707_HOOK_PIN.Error_T1.ET := T#0MS;
   S707_HOOK_PIN.Error_T1.STATE := B#16#0;
   S707_HOOK_PIN.Error_T1.STIME := T#23D5H8M43S363MS;
   S707_HOOK_PIN.Error_T1.ATIME := T#23D5H8M43S986MS;
   S707_HOOK_PIN.Error_T2.IN := FALSE;
   S707_HOOK_PIN.Error_T2.PT := T#4S;
   S707_HOOK_PIN.Error_T2.Q := FALSE;
   S707_HOOK_PIN.Error_T2.ET := T#0MS;
   S707_HOOK_PIN.Error_T2.STATE := B#16#0;
   S707_HOOK_PIN.Error_T2.STIME := T#0MS;
   S707_HOOK_PIN.Error_T2.ATIME := T#0MS;
   S707_HOOK_PIN.CHK_Aux1 := FALSE;
   S707_HOOK_PIN.CHK_Aux2 := FALSE;
   S707_HOOK_PIN.Error_T1_DN := FALSE;
   S707_HOOK_PIN.Error_T2_DN := FALSE;
   S707_HOOK_PIN.Adv_Memo := FALSE;
   S707_HOOK_PIN.Visu_Adv_Arr[0] := FALSE;
   S707_HOOK_PIN.Visu_Adv_Arr[1] := FALSE;
   S707_HOOK_PIN.Visu_Adv_Arr[2] := FALSE;
   S707_HOOK_PIN.Visu_Adv_Arr[3] := FALSE;
   S707_HOOK_PIN.Visu_Adv_Arr[4] := FALSE;
   S707_HOOK_PIN.Visu_Adv_Arr[5] := FALSE;
   S707_HOOK_PIN.Visu_Adv_Arr[6] := FALSE;
   S707_HOOK_PIN.Visu_Adv_Arr[7] := FALSE;
   S707_HOOK_PIN.Visu_Adv_Arr[8] := FALSE;
   S707_HOOK_PIN.Visu_Adv_Arr[9] := FALSE;
   S707_HOOK_PIN.Visu_Adv_Arr[10] := FALSE;
   S707_HOOK_PIN.Visu_Adv_Arr[11] := FALSE;
   S707_HOOK_PIN.Visu_Adv_Arr[12] := FALSE;
   S707_HOOK_PIN.Visu_Adv_Arr[13] := FALSE;
   S707_HOOK_PIN.Visu_Adv_Arr[14] := FALSE;
   S707_HOOK_PIN.Visu_Adv_Arr[15] := FALSE;
   S707_HOOK_PIN.Visu_Ret_Arr[0] := TRUE;
   S707_HOOK_PIN.Visu_Ret_Arr[1] := TRUE;
   S707_HOOK_PIN.Visu_Ret_Arr[2] := TRUE;
   S707_HOOK_PIN.Visu_Ret_Arr[3] := FALSE;
   S707_HOOK_PIN.Visu_Ret_Arr[4] := FALSE;
   S707_HOOK_PIN.Visu_Ret_Arr[5] := FALSE;
   S707_HOOK_PIN.Visu_Ret_Arr[6] := FALSE;
   S707_HOOK_PIN.Visu_Ret_Arr[7] := FALSE;
   S707_HOOK_PIN.Visu_Ret_Arr[8] := FALSE;
   S707_HOOK_PIN.Visu_Ret_Arr[9] := FALSE;
   S707_HOOK_PIN.Visu_Ret_Arr[10] := FALSE;
   S707_HOOK_PIN.Visu_Ret_Arr[11] := FALSE;
   S707_HOOK_PIN.Visu_Ret_Arr[12] := FALSE;
   S707_HOOK_PIN.Visu_Ret_Arr[13] := FALSE;
   S707_HOOK_PIN.Visu_Ret_Arr[14] := FALSE;
   S707_HOOK_PIN.Visu_Ret_Arr[15] := FALSE;
   S707_HOOK_PIN.BLK_Move_Ret := 0;
   S707_HOOK_PIN.Enable := TRUE;
   S707_HOOK_PIN.Adv_End := FALSE;
   S707_HOOK_PIN.Ret_End := TRUE;
   S707_DEACHA_LOCK.Enable_Aux := TRUE;
   S707_DEACHA_LOCK.Adv_Amount := 1;
   S707_DEACHA_LOCK.Ret_Amount := 1;
   S707_DEACHA_LOCK.LS_Adv1 := TRUE;
   S707_DEACHA_LOCK.LS_Ret1 := FALSE;
   S707_DEACHA_LOCK.LS_Adv2 := FALSE;
   S707_DEACHA_LOCK.LS_Ret2 := FALSE;
   S707_DEACHA_LOCK.LS_Adv3 := FALSE;
   S707_DEACHA_LOCK.LS_Ret3 := FALSE;
   S707_DEACHA_LOCK.LS_Adv4 := FALSE;
   S707_DEACHA_LOCK.LS_Ret4 := FALSE;
   S707_DEACHA_LOCK.SOL_Adv := FALSE;
   S707_DEACHA_LOCK.SOL_Ret := FALSE;
   S707_DEACHA_LOCK.M_Ready := TRUE;
   S707_DEACHA_LOCK.T_CHK1 := T#4S;
   S707_DEACHA_LOCK.T_CHK2 := T#4S;
   S707_DEACHA_LOCK.PB_Lamp_CHK := FALSE;
   S707_DEACHA_LOCK.PB_Error_Rst := FALSE;
   S707_DEACHA_LOCK.M_FLICK := FALSE;
   S707_DEACHA_LOCK.M_Adv_Err := FALSE;
   S707_DEACHA_LOCK.M_Ret_Err := FALSE;
   S707_DEACHA_LOCK.LP_Adv := TRUE;
   S707_DEACHA_LOCK.LP_Ret := FALSE;
   S707_DEACHA_LOCK.Visu_Adv := W#16#300;
   S707_DEACHA_LOCK.Visu_Ret := W#16#0;
   S707_DEACHA_LOCK.Error_T1.IN := FALSE;
   S707_DEACHA_LOCK.Error_T1.PT := T#4S;
   S707_DEACHA_LOCK.Error_T1.Q := FALSE;
   S707_DEACHA_LOCK.Error_T1.ET := T#0MS;
   S707_DEACHA_LOCK.Error_T1.STATE := B#16#0;
   S707_DEACHA_LOCK.Error_T1.STIME := T#23D5H8M43S363MS;
   S707_DEACHA_LOCK.Error_T1.ATIME := T#23D5H8M44S238MS;
   S707_DEACHA_LOCK.Error_T2.IN := FALSE;
   S707_DEACHA_LOCK.Error_T2.PT := T#4S;
   S707_DEACHA_LOCK.Error_T2.Q := FALSE;
   S707_DEACHA_LOCK.Error_T2.ET := T#0MS;
   S707_DEACHA_LOCK.Error_T2.STATE := B#16#0;
   S707_DEACHA_LOCK.Error_T2.STIME := T#0MS;
   S707_DEACHA_LOCK.Error_T2.ATIME := T#0MS;
   S707_DEACHA_LOCK.CHK_Aux1 := FALSE;
   S707_DEACHA_LOCK.CHK_Aux2 := FALSE;
   S707_DEACHA_LOCK.Error_T1_DN := FALSE;
   S707_DEACHA_LOCK.Error_T2_DN := FALSE;
   S707_DEACHA_LOCK.Adv_Memo := TRUE;
   S707_DEACHA_LOCK.Visu_Adv_Arr[0] := TRUE;
   S707_DEACHA_LOCK.Visu_Adv_Arr[1] := TRUE;
   S707_DEACHA_LOCK.Visu_Adv_Arr[2] := FALSE;
   S707_DEACHA_LOCK.Visu_Adv_Arr[3] := FALSE;
   S707_DEACHA_LOCK.Visu_Adv_Arr[4] := FALSE;
   S707_DEACHA_LOCK.Visu_Adv_Arr[5] := FALSE;
   S707_DEACHA_LOCK.Visu_Adv_Arr[6] := FALSE;
   S707_DEACHA_LOCK.Visu_Adv_Arr[7] := FALSE;
   S707_DEACHA_LOCK.Visu_Adv_Arr[8] := FALSE;
   S707_DEACHA_LOCK.Visu_Adv_Arr[9] := FALSE;
   S707_DEACHA_LOCK.Visu_Adv_Arr[10] := FALSE;
   S707_DEACHA_LOCK.Visu_Adv_Arr[11] := FALSE;
   S707_DEACHA_LOCK.Visu_Adv_Arr[12] := FALSE;
   S707_DEACHA_LOCK.Visu_Adv_Arr[13] := FALSE;
   S707_DEACHA_LOCK.Visu_Adv_Arr[14] := FALSE;
   S707_DEACHA_LOCK.Visu_Adv_Arr[15] := FALSE;
   S707_DEACHA_LOCK.Visu_Ret_Arr[0] := FALSE;
   S707_DEACHA_LOCK.Visu_Ret_Arr[1] := FALSE;
   S707_DEACHA_LOCK.Visu_Ret_Arr[2] := FALSE;
   S707_DEACHA_LOCK.Visu_Ret_Arr[3] := FALSE;
   S707_DEACHA_LOCK.Visu_Ret_Arr[4] := FALSE;
   S707_DEACHA_LOCK.Visu_Ret_Arr[5] := FALSE;
   S707_DEACHA_LOCK.Visu_Ret_Arr[6] := FALSE;
   S707_DEACHA_LOCK.Visu_Ret_Arr[7] := FALSE;
   S707_DEACHA_LOCK.Visu_Ret_Arr[8] := FALSE;
   S707_DEACHA_LOCK.Visu_Ret_Arr[9] := FALSE;
   S707_DEACHA_LOCK.Visu_Ret_Arr[10] := FALSE;
   S707_DEACHA_LOCK.Visu_Ret_Arr[11] := FALSE;
   S707_DEACHA_LOCK.Visu_Ret_Arr[12] := FALSE;
   S707_DEACHA_LOCK.Visu_Ret_Arr[13] := FALSE;
   S707_DEACHA_LOCK.Visu_Ret_Arr[14] := FALSE;
   S707_DEACHA_LOCK.Visu_Ret_Arr[15] := FALSE;
   S707_DEACHA_LOCK.BLK_Move_Ret := 0;
   S707_DEACHA_LOCK.Enable := TRUE;
   S707_DEACHA_LOCK.Adv_End := TRUE;
   S707_DEACHA_LOCK.Ret_End := FALSE;
   S707_ELE.Enable_Aux := TRUE;
   S707_ELE.Adv_Amount := 1;
   S707_ELE.Ret_Amount := 1;
   S707_ELE.LS_Adv1 := TRUE;
   S707_ELE.LS_Ret1 := FALSE;
   S707_ELE.LS_Adv2 := FALSE;
   S707_ELE.LS_Ret2 := FALSE;
   S707_ELE.LS_Adv3 := FALSE;
   S707_ELE.LS_Ret3 := FALSE;
   S707_ELE.LS_Adv4 := FALSE;
   S707_ELE.LS_Ret4 := FALSE;
   S707_ELE.SOL_Adv := FALSE;
   S707_ELE.SOL_Ret := FALSE;
   S707_ELE.M_Ready := TRUE;
   S707_ELE.T_CHK1 := T#4S;
   S707_ELE.T_CHK2 := T#4S;
   S707_ELE.PB_Lamp_CHK := FALSE;
   S707_ELE.PB_Error_Rst := FALSE;
   S707_ELE.M_FLICK := FALSE;
   S707_ELE.M_Adv_Err := FALSE;
   S707_ELE.M_Ret_Err := FALSE;
   S707_ELE.LP_Adv := TRUE;
   S707_ELE.LP_Ret := FALSE;
   S707_ELE.Visu_Adv := W#16#300;
   S707_ELE.Visu_Ret := W#16#0;
   S707_ELE.Error_T1.IN := FALSE;
   S707_ELE.Error_T1.PT := T#4S;
   S707_ELE.Error_T1.Q := FALSE;
   S707_ELE.Error_T1.ET := T#0MS;
   S707_ELE.Error_T1.STATE := B#16#0;
   S707_ELE.Error_T1.STIME := T#23D5H8M47S258MS;
   S707_ELE.Error_T1.ATIME := T#23D5H8M47S483MS;
   S707_ELE.Error_T2.IN := FALSE;
   S707_ELE.Error_T2.PT := T#4S;
   S707_ELE.Error_T2.Q := FALSE;
   S707_ELE.Error_T2.ET := T#0MS;
   S707_ELE.Error_T2.STATE := B#16#0;
   S707_ELE.Error_T2.STIME := T#0MS;
   S707_ELE.Error_T2.ATIME := T#0MS;
   S707_ELE.CHK_Aux1 := FALSE;
   S707_ELE.CHK_Aux2 := FALSE;
   S707_ELE.Error_T1_DN := FALSE;
   S707_ELE.Error_T2_DN := FALSE;
   S707_ELE.Adv_Memo := TRUE;
   S707_ELE.Visu_Adv_Arr[0] := TRUE;
   S707_ELE.Visu_Adv_Arr[1] := TRUE;
   S707_ELE.Visu_Adv_Arr[2] := FALSE;
   S707_ELE.Visu_Adv_Arr[3] := FALSE;
   S707_ELE.Visu_Adv_Arr[4] := FALSE;
   S707_ELE.Visu_Adv_Arr[5] := FALSE;
   S707_ELE.Visu_Adv_Arr[6] := FALSE;
   S707_ELE.Visu_Adv_Arr[7] := FALSE;
   S707_ELE.Visu_Adv_Arr[8] := FALSE;
   S707_ELE.Visu_Adv_Arr[9] := FALSE;
   S707_ELE.Visu_Adv_Arr[10] := FALSE;
   S707_ELE.Visu_Adv_Arr[11] := FALSE;
   S707_ELE.Visu_Adv_Arr[12] := FALSE;
   S707_ELE.Visu_Adv_Arr[13] := FALSE;
   S707_ELE.Visu_Adv_Arr[14] := FALSE;
   S707_ELE.Visu_Adv_Arr[15] := FALSE;
   S707_ELE.Visu_Ret_Arr[0] := FALSE;
   S707_ELE.Visu_Ret_Arr[1] := FALSE;
   S707_ELE.Visu_Ret_Arr[2] := FALSE;
   S707_ELE.Visu_Ret_Arr[3] := FALSE;
   S707_ELE.Visu_Ret_Arr[4] := FALSE;
   S707_ELE.Visu_Ret_Arr[5] := FALSE;
   S707_ELE.Visu_Ret_Arr[6] := FALSE;
   S707_ELE.Visu_Ret_Arr[7] := FALSE;
   S707_ELE.Visu_Ret_Arr[8] := FALSE;
   S707_ELE.Visu_Ret_Arr[9] := FALSE;
   S707_ELE.Visu_Ret_Arr[10] := FALSE;
   S707_ELE.Visu_Ret_Arr[11] := FALSE;
   S707_ELE.Visu_Ret_Arr[12] := FALSE;
   S707_ELE.Visu_Ret_Arr[13] := FALSE;
   S707_ELE.Visu_Ret_Arr[14] := FALSE;
   S707_ELE.Visu_Ret_Arr[15] := FALSE;
   S707_ELE.BLK_Move_Ret := 0;
   S707_ELE.Enable := TRUE;
   S707_ELE.Adv_End := TRUE;
   S707_ELE.Ret_End := FALSE;
   S707_AIR_ELE.Enable_Aux := TRUE;
   S707_AIR_ELE.Adv_Amount := 1;
   S707_AIR_ELE.Ret_Amount := 1;
   S707_AIR_ELE.LS_Adv1 := TRUE;
   S707_AIR_ELE.LS_Ret1 := FALSE;
   S707_AIR_ELE.LS_Adv2 := FALSE;
   S707_AIR_ELE.LS_Ret2 := FALSE;
   S707_AIR_ELE.LS_Adv3 := FALSE;
   S707_AIR_ELE.LS_Ret3 := FALSE;
   S707_AIR_ELE.LS_Adv4 := FALSE;
   S707_AIR_ELE.LS_Ret4 := FALSE;
   S707_AIR_ELE.SOL_Adv := FALSE;
   S707_AIR_ELE.SOL_Ret := FALSE;
   S707_AIR_ELE.M_Ready := TRUE;
   S707_AIR_ELE.T_CHK1 := T#4S;
   S707_AIR_ELE.T_CHK2 := T#4S;
   S707_AIR_ELE.PB_Lamp_CHK := FALSE;
   S707_AIR_ELE.PB_Error_Rst := FALSE;
   S707_AIR_ELE.M_FLICK := FALSE;
   S707_AIR_ELE.M_Adv_Err := FALSE;
   S707_AIR_ELE.M_Ret_Err := FALSE;
   S707_AIR_ELE.LP_Adv := TRUE;
   S707_AIR_ELE.LP_Ret := FALSE;
   S707_AIR_ELE.Visu_Adv := W#16#300;
   S707_AIR_ELE.Visu_Ret := W#16#0;
   S707_AIR_ELE.Error_T1.IN := FALSE;
   S707_AIR_ELE.Error_T1.PT := T#4S;
   S707_AIR_ELE.Error_T1.Q := FALSE;
   S707_AIR_ELE.Error_T1.ET := T#0MS;
   S707_AIR_ELE.Error_T1.STATE := B#16#0;
   S707_AIR_ELE.Error_T1.STIME := T#23D5H8M47S258MS;
   S707_AIR_ELE.Error_T1.ATIME := T#23D5H8M47S349MS;
   S707_AIR_ELE.Error_T2.IN := FALSE;
   S707_AIR_ELE.Error_T2.PT := T#4S;
   S707_AIR_ELE.Error_T2.Q := FALSE;
   S707_AIR_ELE.Error_T2.ET := T#0MS;
   S707_AIR_ELE.Error_T2.STATE := B#16#0;
   S707_AIR_ELE.Error_T2.STIME := T#0MS;
   S707_AIR_ELE.Error_T2.ATIME := T#0MS;
   S707_AIR_ELE.CHK_Aux1 := FALSE;
   S707_AIR_ELE.CHK_Aux2 := FALSE;
   S707_AIR_ELE.Error_T1_DN := FALSE;
   S707_AIR_ELE.Error_T2_DN := FALSE;
   S707_AIR_ELE.Adv_Memo := TRUE;
   S707_AIR_ELE.Visu_Adv_Arr[0] := TRUE;
   S707_AIR_ELE.Visu_Adv_Arr[1] := TRUE;
   S707_AIR_ELE.Visu_Adv_Arr[2] := FALSE;
   S707_AIR_ELE.Visu_Adv_Arr[3] := FALSE;
   S707_AIR_ELE.Visu_Adv_Arr[4] := FALSE;
   S707_AIR_ELE.Visu_Adv_Arr[5] := FALSE;
   S707_AIR_ELE.Visu_Adv_Arr[6] := FALSE;
   S707_AIR_ELE.Visu_Adv_Arr[7] := FALSE;
   S707_AIR_ELE.Visu_Adv_Arr[8] := FALSE;
   S707_AIR_ELE.Visu_Adv_Arr[9] := FALSE;
   S707_AIR_ELE.Visu_Adv_Arr[10] := FALSE;
   S707_AIR_ELE.Visu_Adv_Arr[11] := FALSE;
   S707_AIR_ELE.Visu_Adv_Arr[12] := FALSE;
   S707_AIR_ELE.Visu_Adv_Arr[13] := FALSE;
   S707_AIR_ELE.Visu_Adv_Arr[14] := FALSE;
   S707_AIR_ELE.Visu_Adv_Arr[15] := FALSE;
   S707_AIR_ELE.Visu_Ret_Arr[0] := FALSE;
   S707_AIR_ELE.Visu_Ret_Arr[1] := FALSE;
   S707_AIR_ELE.Visu_Ret_Arr[2] := FALSE;
   S707_AIR_ELE.Visu_Ret_Arr[3] := FALSE;
   S707_AIR_ELE.Visu_Ret_Arr[4] := FALSE;
   S707_AIR_ELE.Visu_Ret_Arr[5] := FALSE;
   S707_AIR_ELE.Visu_Ret_Arr[6] := FALSE;
   S707_AIR_ELE.Visu_Ret_Arr[7] := FALSE;
   S707_AIR_ELE.Visu_Ret_Arr[8] := FALSE;
   S707_AIR_ELE.Visu_Ret_Arr[9] := FALSE;
   S707_AIR_ELE.Visu_Ret_Arr[10] := FALSE;
   S707_AIR_ELE.Visu_Ret_Arr[11] := FALSE;
   S707_AIR_ELE.Visu_Ret_Arr[12] := FALSE;
   S707_AIR_ELE.Visu_Ret_Arr[13] := FALSE;
   S707_AIR_ELE.Visu_Ret_Arr[14] := FALSE;
   S707_AIR_ELE.Visu_Ret_Arr[15] := FALSE;
   S707_AIR_ELE.BLK_Move_Ret := 0;
   S707_AIR_ELE.Enable := TRUE;
   S707_AIR_ELE.Adv_End := TRUE;
   S707_AIR_ELE.Ret_End := FALSE;
END_DATA_BLOCK

FUNCTION FC 131 : VOID
TITLE =
VERSION : 0.1

BEGIN
NETWORK
TITLE =
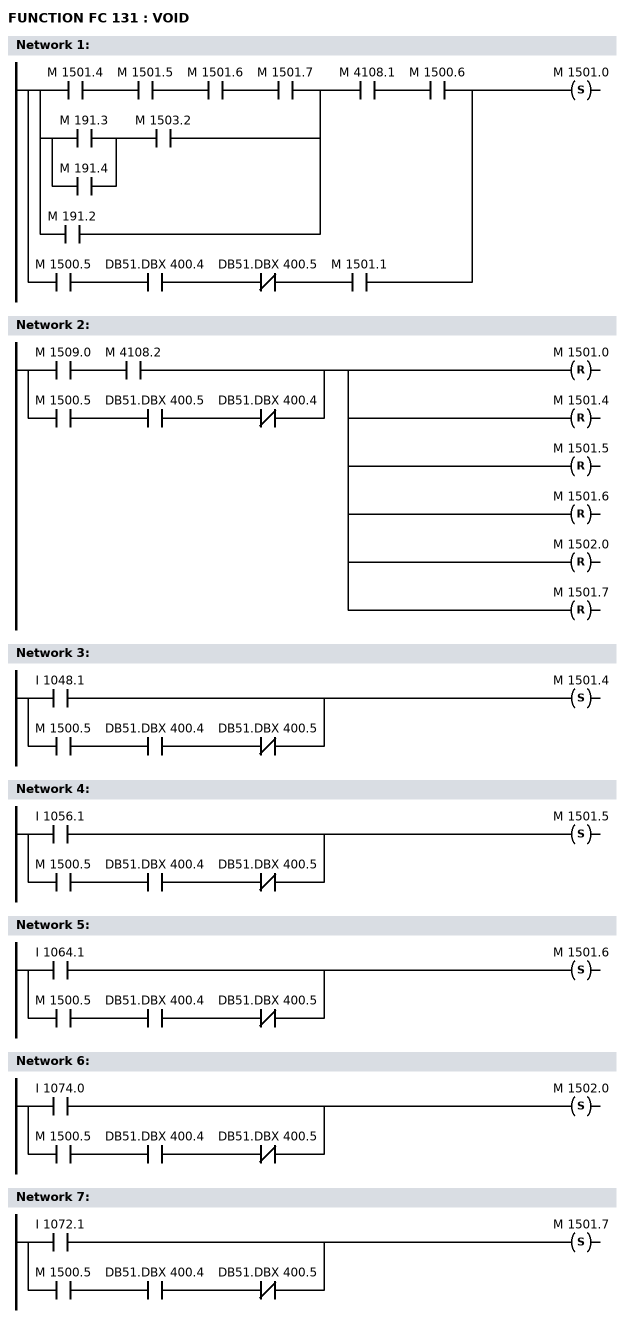

      A(    ;
      A     M   1501.4;
      A     M   1501.5;
      A     M   1501.6;
      A     M   1501.7;
      O     ;
      A(    ;
      O     M    191.3;
      O     M    191.4;
      )     ;
      A     M   1503.2;
      O     M    191.2;
      )     ;
      A     M   4108.1;
      A     M   1500.6;
      O     ;
      A     M   1500.5;
      A     DB51.DBX  400.4;
      AN    DB51.DBX  400.5;
      A     M   1501.1;
      S     M   1501.0;
NETWORK
TITLE =

      A     M   1509.0;
      A     M   4108.2;
      O     ;
      A     M   1500.5;
      A     DB51.DBX  400.5;
      AN    DB51.DBX  400.4;
      R     M   1501.0;
      R     M   1501.4;
      R     M   1501.5;
      R     M   1501.6;
      R     M   1502.0;
      R     M   1501.7;
NETWORK
TITLE =

      O     I   1048.1;
      O     ;
      A     M   1500.5;
      A     DB51.DBX  400.4;
      AN    DB51.DBX  400.5;
      S     M   1501.4;
NETWORK
TITLE =

      O     I   1056.1;
      O     ;
      A     M   1500.5;
      A     DB51.DBX  400.4;
      AN    DB51.DBX  400.5;
      S     M   1501.5;
NETWORK
TITLE =

      O     I   1064.1;
      O     ;
      A     M   1500.5;
      A     DB51.DBX  400.4;
      AN    DB51.DBX  400.5;
      S     M   1501.6;
NETWORK
TITLE =

      O     I   1074.0;
      O     ;
      A     M   1500.5;
      A     DB51.DBX  400.4;
      AN    DB51.DBX  400.5;
      S     M   1502.0;
NETWORK
TITLE =

      O     I   1072.1;
      O     ;
      A     M   1500.5;
      A     DB51.DBX  400.4;
      AN    DB51.DBX  400.5;
      S     M   1501.7;
END_FUNCTION

FUNCTION_BLOCK FB 132
TITLE =
VERSION : 0.1

BEGIN
NETWORK
TITLE =
